LIN {X 0,Y 355.905,Z 472.152,A -85,B 0,C 180,E1 -13283.259,E2 -13283.259} C_VEL
LIN {X 0,Y 354.805,Z 472.289,A -85,B 0,C 180,E1 -13284.204,E2 -13284.204} C_VEL
LIN {X 0,Y 354.689,Z 472.301,A -85,B 0,C 180,E1 -13284.524,E2 -13284.524} C_VEL
LIN {X 0,Y 354.395,Z 472.343,A -85,B 0,C 180,E1 -13287.626,E2 -13287.626} C_VEL
LIN {X 0,Y 353.979,Z 472.396,A -85,B 0,C 180,E1 -13291.542,E2 -13291.542} C_VEL
LIN {X 0,Y 353.842,Z 472.551,A -85,B 0,C 180,E1 -13292.817,E2 -13292.817} C_VEL
LIN {X 0,Y 353.738,Z 476.121,A -85,B 0,C 180,E1 -13296.587,E2 -13296.587} C_VEL
LIN {X 0,Y 353.621,Z 479.721,A -85,B 0,C 180,E1 -13300.253,E2 -13300.253} C_VEL
LIN {X 0,Y 353.632,Z 480.392,A -85,B 0,C 180,E1 -13300.924,E2 -13300.924} C_VEL
LIN {X 0,Y 356.212,Z 492.931,A -85,B 0,C 180,E1 -13301.598,E2 -13301.598} C_VEL
LIN {X 0,Y 359.042,Z 506.674,A -85,B 0,C 180,E1 -13302.568,E2 -13302.568} C_VEL
LIN {X 0,Y 358.364,Z 517.999,A -85,B 0,C 180,E1 -13303.479,E2 -13303.479} C_VEL
LIN {X 0,Y 357.519,Z 529.506,A -85,B 0,C 180,E1 -13304.642,E2 -13304.642} C_VEL
LIN {X 0,Y 356.647,Z 540.627,A -85,B 0,C 180,E1 -13306.031,E2 -13306.031} C_VEL
LIN {X 0,Y 355.769,Z 549.851,A -85,B 0,C 180,E1 -13307.449,E2 -13307.449} C_VEL
LIN {X 0,Y 355.032,Z 558.925,A -85,B 0,C 180,E1 -13309.16,E2 -13309.16} C_VEL
LIN {X 0,Y 354.441,Z 566.279,A -85,B 0,C 180,E1 -13310.873,E2 -13310.873} C_VEL
LIN {X 0,Y 354.04,Z 572.161,A -85,B 0,C 180,E1 -13312.587,E2 -13312.587} C_VEL
LIN {X 0,Y 353.758,Z 576.815,A -85,B 0,C 180,E1 -13314.299,E2 -13314.299} C_VEL
LIN {X 0,Y 353.549,Z 580.37,A -85,B 0,C 180,E1 -13316.01,E2 -13316.01} C_VEL
LIN {X 0,Y 353.522,Z 582.903,A -85,B 0,C 180,E1 -13317.721,E2 -13317.721} C_VEL
LIN {X 0,Y 353.486,Z 584.043,A -85,B 0,C 180,E1 -13318.861,E2 -13318.861} C_VEL
LIN {X 0,Y 353.456,Z 584.785,A -85,B 0,C 180,E1 -13320,E2 -13320} C_VEL
LIN {X 0,Y 353.525,Z 585.12,A -85,B 0,C 180,E1 -13321.139,E2 -13321.139} C_VEL
LIN {X 0,Y 353.644,Z 585.007,A -85,B 0,C 180,E1 -13322.278,E2 -13322.278} C_VEL
LIN {X 0,Y 353.82,Z 584.499,A -85,B 0,C 180,E1 -13323.416,E2 -13323.416} C_VEL
LIN {X 0,Y 354.023,Z 583.603,A -85,B 0,C 180,E1 -13324.554,E2 -13324.554} C_VEL
LIN {X 0,Y 354.055,Z 582.303,A -85,B 0,C 180,E1 -13325.696,E2 -13325.696} C_VEL
LIN {X 0,Y 354.716,Z 578.614,A -85,B 0,C 180,E1 -13327.838,E2 -13327.838} C_VEL
LIN {X 0,Y 355.446,Z 574.19,A -85,B 0,C 180,E1 -13329.675,E2 -13329.675} C_VEL
LIN {X 0,Y 356.568,Z 567.89,A -85,B 0,C 180,E1 -13331.655,E2 -13331.655} C_VEL
LIN {X 0,Y 357.659,Z 561.049,A -85,B 0,C 180,E1 -13333.349,E2 -13333.349} C_VEL
LIN {X 0,Y 358.995,Z 552.647,A -85,B 0,C 180,E1 -13335.034,E2 -13335.034} C_VEL
LIN {X 0,Y 360.549,Z 544.142,A -85,B 0,C 180,E1 -13336.418,E2 -13336.418} C_VEL
LIN {X 0,Y 362.18,Z 532.806,A -85,B 0,C 180,E1 -13337.931,E2 -13337.931} C_VEL
LIN {X 0,Y 363.831,Z 521.052,A -85,B 0,C 180,E1 -13339.171,E2 -13339.171} C_VEL
LIN {X 0,Y 364.531,Z 514.204,A -85,B 0,C 180,E1 -13339.791,E2 -13339.791} C_VEL
LIN {X 0,Y 362.046,Z 504.538,A -85,B 0,C 180,E1 -13340.902,E2 -13340.902} C_VEL
LIN {X 0,Y 358.084,Z 494.328,A -85,B 0,C 180,E1 -13342.101,E2 -13342.101} C_VEL
LIN {X 0,Y 355.734,Z 489.62,A -85,B 0,C 180,E1 -13342.687,E2 -13342.687} C_VEL
LIN {X 0,Y 354.862,Z 487.017,A -85,B 0,C 180,E1 -13342.988,E2 -13342.988} C_VEL
LIN {X 0,Y 355.255,Z 485.091,A -85,B 0,C 180,E1 -13347.065,E2 -13347.065} C_VEL
LIN {X 0,Y 355.732,Z 483.771,A -85,B 0,C 180,E1 -13350.908,E2 -13350.908} C_VEL
LIN {X 0,Y 356.135,Z 483.121,A -85,B 0,C 180,E1 -13354.021,E2 -13354.021} C_VEL
LIN {X 0,Y 356.41,Z 482.934,A -85,B 0,C 180,E1 -13356.268,E2 -13356.268} C_VEL
LIN {X 0,Y 356.662,Z 483.11,A -85,B 0,C 180,E1 -13359.091,E2 -13359.091} C_VEL
LIN {X 0,Y 356.824,Z 483.837,A -85,B 0,C 180,E1 -13362.041,E2 -13362.041} C_VEL
LIN {X 0,Y 357.107,Z 485.188,A -85,B 0,C 180,E1 -13365.112,E2 -13365.112} C_VEL
LIN {X 0,Y 357.505,Z 487.296,A -85,B 0,C 180,E1 -13368.333,E2 -13368.333} C_VEL
LIN {X 0,Y 357.859,Z 490.386,A -85,B 0,C 180,E1 -13371.773,E2 -13371.773} C_VEL
LIN {X 0,Y 357.766,Z 492.788,A -85,B 0,C 180,E1 -13373.891,E2 -13373.891} C_VEL
LIN {X 0,Y 357.119,Z 496.371,A -85,B 0,C 180,E1 -13376.562,E2 -13376.562} C_VEL
LIN {X 0,Y 356.022,Z 502.317,A -85,B 0,C 180,E1 -13380.428,E2 -13380.428} C_VEL
LIN {X 0,Y 355.137,Z 508.799,A -85,B 0,C 180,E1 -13384.191,E2 -13384.191} C_VEL
LIN {X 0,Y 354.64,Z 514.033,A -85,B 0,C 180,E1 -13386.959,E2 -13386.959} C_VEL
LIN {X 0,Y 355.608,Z 517.659,A -85,B 0,C 180,E1 -13387.26,E2 -13387.26} C_VEL
LIN {X 0,Y 358.687,Z 529.151,A -85,B 0,C 180,E1 -13388.286,E2 -13388.286} C_VEL
LIN {X 0,Y 360.594,Z 540.569,A -85,B 0,C 180,E1 -13389.313,E2 -13389.313} C_VEL
LIN {X 0,Y 361.291,Z 549.72,A -85,B 0,C 180,E1 -13390.174,E2 -13390.174} C_VEL
LIN {X 0,Y 360.953,Z 561.989,A -85,B 0,C 180,E1 -13391.408,E2 -13391.408} C_VEL
LIN {X 0,Y 359.23,Z 574.08,A -85,B 0,C 180,E1 -13392.788,E2 -13392.788} C_VEL
LIN {X 0,Y 357.65,Z 584.49,A -85,B 0,C 180,E1 -13394.251,E2 -13394.251} C_VEL
LIN {X 0,Y 356.354,Z 593.147,A -85,B 0,C 180,E1 -13395.728,E2 -13395.728} C_VEL
LIN {X 0,Y 355.292,Z 601.393,A -85,B 0,C 180,E1 -13397.432,E2 -13397.432} C_VEL
LIN {X 0,Y 354.388,Z 608.162,A -85,B 0,C 180,E1 -13399.141,E2 -13399.141} C_VEL
LIN {X 0,Y 353.849,Z 613.658,A -85,B 0,C 180,E1 -13400.857,E2 -13400.857} C_VEL
LIN {X 0,Y 353.509,Z 618,A -85,B 0,C 180,E1 -13402.575,E2 -13402.575} C_VEL
LIN {X 0,Y 353.335,Z 621.292,A -85,B 0,C 180,E1 -13404.292,E2 -13404.292} C_VEL
LIN {X 0,Y 353.326,Z 622.934,A -85,B 0,C 180,E1 -13405.436,E2 -13405.436} C_VEL
LIN {X 0,Y 353.371,Z 624.929,A -85,B 0,C 180,E1 -13407.72,E2 -13407.72} C_VEL
LIN {X 0,Y 353.465,Z 625.318,A -85,B 0,C 180,E1 -13408.861,E2 -13408.861} C_VEL
LIN {X 0,Y 353.463,Z 625.241,A -85,B 0,C 180,E1 -13410,E2 -13410} C_VEL
LIN {X 0,Y 353.476,Z 624.735,A -85,B 0,C 180,E1 -13411.139,E2 -13411.139} C_VEL
LIN {X 0,Y 353.477,Z 623.816,A -85,B 0,C 180,E1 -13412.279,E2 -13412.279} C_VEL
LIN {X 0,Y 353.344,Z 622.452,A -85,B 0,C 180,E1 -13413.421,E2 -13413.421} C_VEL
LIN {X 0,Y 353.457,Z 619.538,A -85,B 0,C 180,E1 -13415.133,E2 -13415.133} C_VEL
LIN {X 0,Y 353.501,Z 615.509,A -85,B 0,C 180,E1 -13416.851,E2 -13416.851} C_VEL
LIN {X 0,Y 353.764,Z 609.258,A -85,B 0,C 180,E1 -13418.857,E2 -13418.857} C_VEL
LIN {X 0,Y 354.144,Z 602.428,A -85,B 0,C 180,E1 -13420.577,E2 -13420.577} C_VEL
LIN {X 0,Y 354.86,Z 593.944,A -85,B 0,C 180,E1 -13422.292,E2 -13422.292} C_VEL
LIN {X 0,Y 355.702,Z 583.664,A -85,B 0,C 180,E1 -13423.958,E2 -13423.958} C_VEL
LIN {X 0,Y 356.569,Z 573.529,A -85,B 0,C 180,E1 -13425.285,E2 -13425.285} C_VEL
LIN {X 0,Y 357.601,Z 561.386,A -85,B 0,C 180,E1 -13426.557,E2 -13426.557} C_VEL
LIN {X 0,Y 357.936,Z 554.907,A -85,B 0,C 180,E1 -13427.129,E2 -13427.129} C_VEL
LIN {X 0,Y 356.748,Z 542.906,A -85,B 0,C 180,E1 -13428.045,E2 -13428.045} C_VEL
LIN {X 0,Y 355.075,Z 528.958,A -85,B 0,C 180,E1 -13428.876,E2 -13428.876} C_VEL
LIN {X 0,Y 353.997,Z 519.742,A -85,B 0,C 180,E1 -13429.31,E2 -13429.31} C_VEL
LIN {X 0,Y 354.501,Z 511.518,A -85,B 0,C 180,E1 -13433.36,E2 -13433.36} C_VEL
LIN {X 0,Y 355.211,Z 504.084,A -85,B 0,C 180,E1 -13437.083,E2 -13437.083} C_VEL
LIN {X 0,Y 355.831,Z 497.874,A -85,B 0,C 180,E1 -13440.241,E2 -13440.241} C_VEL
LIN {X 0,Y 356.571,Z 491.594,A -85,B 0,C 180,E1 -13443.496,E2 -13443.496} C_VEL
LIN {X 0,Y 356.992,Z 487.823,A -85,B 0,C 180,E1 -13445.504,E2 -13445.504} C_VEL
LIN {X 0,Y 356.888,Z 483.993,A -85,B 0,C 180,E1 -13447.623,E2 -13447.623} C_VEL
LIN {X 0,Y 356.029,Z 478.756,A -85,B 0,C 180,E1 -13450.649,E2 -13450.649} C_VEL
LIN {X 0,Y 354.875,Z 472.282,A -85,B 0,C 180,E1 -13454.685,E2 -13454.685} C_VEL
LIN {X 0,Y 354.838,Z 472.282,A -85,B 0,C 180,E1 -13457.669,E2 -13457.669} C_VEL
LIN {X 0,Y 354.821,Z 472.289,A -85,B 0,C 180,E1 -13460.667,E2 -13460.667} C_VEL
LIN {X 0,Y 354.822,Z 472.287,A -85,B 0,C 180,E1 -13464.301,E2 -13464.301} C_VEL
LIN {X 0,Y 354.788,Z 472.288,A -85,B 0,C 180,E1 -13467.667,E2 -13467.667} C_VEL
LIN {X 0,Y 354.847,Z 472.281,A -85,B 0,C 180,E1 -13471.619,E2 -13471.619} C_VEL
LIN {X 0,Y 354.9,Z 472.276,A -85,B 0,C 180,E1 -13474.173,E2 -13474.173} C_VEL
LIN {X 0,Y 354.836,Z 472.283,A -85,B 0,C 180,E1 -13477.894,E2 -13477.894} C_VEL
LIN {X 0,Y 354.923,Z 472.272,A -85,B 0,C 180,E1 -13481.892,E2 -13481.892} C_VEL
LIN {X 0,Y 354.944,Z 472.27,A -85,B 0,C 180,E1 -13485.981,E2 -13485.981} C_VEL
LIN {X 0,Y 354.98,Z 472.264,A -85,B 0,C 180,E1 -13489.736,E2 -13489.736} C_VEL
LIN {X 0,Y 355.116,Z 472.249,A -85,B 0,C 180,E1 -13492.037,E2 -13492.037} C_VEL
LIN {X 0,Y 355.094,Z 472.255,A -85,B 0,C 180,E1 -13494.321,E2 -13494.321} C_VEL
LIN {X 0,Y 355.245,Z 472.231,A -85,B 0,C 180,E1 -13497.733,E2 -13497.733} C_VEL
LIN {X 0,Y 355.4,Z 472.214,A -85,B 0,C 180,E1 -13500,E2 -13500} C_VEL
LIN {X 0,Y 355.247,Z 472.235,A -85,B 0,C 180,E1 -13502.268,E2 -13502.268} C_VEL
LIN {X 0,Y 355.14,Z 472.248,A -85,B 0,C 180,E1 -13506.819,E2 -13506.819} C_VEL
LIN {X 0,Y 355.017,Z 472.261,A -85,B 0,C 180,E1 -13509.113,E2 -13509.113} C_VEL
LIN {X 0,Y 354.924,Z 472.276,A -85,B 0,C 180,E1 -13512.581,E2 -13512.581} C_VEL
LIN {X 0,Y 354.892,Z 472.279,A -85,B 0,C 180,E1 -13516.096,E2 -13516.096} C_VEL
LIN {X 0,Y 354.908,Z 472.278,A -85,B 0,C 180,E1 -13518.472,E2 -13518.472} C_VEL
LIN {X 0,Y 354.837,Z 472.286,A -85,B 0,C 180,E1 -13522.106,E2 -13522.106} C_VEL
LIN {X 0,Y 354.902,Z 472.276,A -85,B 0,C 180,E1 -13525.828,E2 -13525.828} C_VEL
LIN {X 0,Y 354.856,Z 472.281,A -85,B 0,C 180,E1 -13529.679,E2 -13529.679} C_VEL
LIN {X 0,Y 354.808,Z 472.286,A -85,B 0,C 180,E1 -13533.702,E2 -13533.702} C_VEL
LIN {X 0,Y 354.801,Z 472.292,A -85,B 0,C 180,E1 -13536.46,E2 -13536.46} C_VEL
LIN {X 0,Y 354.826,Z 472.284,A -85,B 0,C 180,E1 -13539.424,E2 -13539.424} C_VEL
LIN {X 0,Y 354.791,Z 472.289,A -85,B 0,C 180,E1 -13542.868,E2 -13542.868} C_VEL
LIN {X 0,Y 354.771,Z 472.295,A -85,B 0,C 180,E1 -13546.104,E2 -13546.104} C_VEL
LIN {X 0,Y 354.791,Z 472.288,A -85,B 0,C 180,E1 -13549.179,E2 -13549.179} C_VEL
LIN {X 0,Y 354.815,Z 472.289,A -85,B 0,C 180,E1 -13552.402,E2 -13552.402} C_VEL
LIN {X 0,Y 354.815,Z 472.285,A -85,B 0,C 180,E1 -13554.941,E2 -13554.941} C_VEL
LIN {X 0,Y 354.797,Z 472.292,A -85,B 0,C 180,E1 -13558.405,E2 -13558.405} C_VEL
LIN {X 0,Y 354.85,Z 472.282,A -85,B 0,C 180,E1 -13561.619,E2 -13561.619} C_VEL
LIN {X 0,Y 354.903,Z 472.279,A -85,B 0,C 180,E1 -13564.173,E2 -13564.173} C_VEL
LIN {X 0,Y 354.838,Z 472.286,A -85,B 0,C 180,E1 -13567.894,E2 -13567.894} C_VEL
LIN {X 0,Y 354.927,Z 472.275,A -85,B 0,C 180,E1 -13571.892,E2 -13571.892} C_VEL
LIN {X 0,Y 354.947,Z 472.273,A -85,B 0,C 180,E1 -13575.981,E2 -13575.981} C_VEL
LIN {X 0,Y 354.982,Z 472.267,A -85,B 0,C 180,E1 -13579.736,E2 -13579.736} C_VEL
LIN {X 0,Y 355.107,Z 472.249,A -85,B 0,C 180,E1 -13583.18,E2 -13583.18} C_VEL
LIN {X 0,Y 355.248,Z 472.235,A -85,B 0,C 180,E1 -13587.733,E2 -13587.733} C_VEL
LIN {X 0,Y 355.401,Z 472.217,A -85,B 0,C 180,E1 -13590,E2 -13590} C_VEL
LIN {X 0,Y 355.248,Z 472.235,A -85,B 0,C 180,E1 -13592.268,E2 -13592.268} C_VEL
LIN {X 0,Y 355.126,Z 472.246,A -85,B 0,C 180,E1 -13596.82,E2 -13596.82} C_VEL
LIN {X 0,Y 354.982,Z 472.267,A -85,B 0,C 180,E1 -13600.264,E2 -13600.264} C_VEL
LIN {X 0,Y 354.947,Z 472.274,A -85,B 0,C 180,E1 -13604.019,E2 -13604.019} C_VEL
LIN {X 0,Y 354.927,Z 472.275,A -85,B 0,C 180,E1 -13608.109,E2 -13608.109} C_VEL
LIN {X 0,Y 354.839,Z 472.286,A -85,B 0,C 180,E1 -13612.106,E2 -13612.106} C_VEL
LIN {X 0,Y 354.903,Z 472.279,A -85,B 0,C 180,E1 -13615.827,E2 -13615.827} C_VEL
LIN {X 0,Y 354.821,Z 472.288,A -85,B 0,C 180,E1 -13619.682,E2 -13619.682} C_VEL
LIN {X 0,Y 354.81,Z 472.291,A -85,B 0,C 180,E1 -13623.702,E2 -13623.702} C_VEL
LIN {X 0,Y 354.802,Z 472.287,A -85,B 0,C 180,E1 -13626.459,E2 -13626.459} C_VEL
LIN {X 0,Y 354.828,Z 472.286,A -85,B 0,C 180,E1 -13629.424,E2 -13629.424} C_VEL
LIN {X 0,Y 354.792,Z 472.288,A -85,B 0,C 180,E1 -13632.867,E2 -13632.867} C_VEL
LIN {X 0,Y 354.771,Z 472.293,A -85,B 0,C 180,E1 -13636.104,E2 -13636.104} C_VEL
LIN {X 0,Y 354.78,Z 472.288,A -85,B 0,C 180,E1 -13639.597,E2 -13639.597} C_VEL
LIN {X 0,Y 354.793,Z 472.288,A -85,B 0,C 180,E1 -13642.406,E2 -13642.406} C_VEL
LIN {X 0,Y 354.689,Z 472.301,A -85,B 0,C 180,E1 -13644.524,E2 -13644.524} C_VEL
LIN {X 0,Y 353.912,Z 472.402,A -85,B 0,C 180,E1 -13645.47,E2 -13645.47} C_VEL
LIN {X 0,Y 350.871,Z 472.777,A -85,B 0,C 180,E1 -13647.002,E2 -13647.002} C_VEL
LIN {X 0,Y 348.33,Z 473.095,A -85,B 0,C 180,E1 -13648.243,E2 -13648.243} C_VEL
LIN {X 0,Y 347.232,Z 473.232,A -85,B 0,C 180,E1 -13649.206,E2 -13649.206} C_VEL
LIN {X 0,Y 347.137,Z 473.246,A -85,B 0,C 180,E1 -13649.533,E2 -13649.533} C_VEL
LIN {X 0,Y 346.856,Z 473.284,A -85,B 0,C 180,E1 -13652.223,E2 -13652.223} C_VEL
LIN {X 0,Y 346.776,Z 473.898,A -85,B 0,C 180,E1 -13653.521,E2 -13653.521} C_VEL
LIN {X 0,Y 346.629,Z 477.509,A -85,B 0,C 180,E1 -13657.342,E2 -13657.342} C_VEL
LIN {X 0,Y 346.574,Z 480.732,A -85,B 0,C 180,E1 -13660.644,E2 -13660.644} C_VEL
LIN {X 0,Y 349.725,Z 496.151,A -85,B 0,C 180,E1 -13661.547,E2 -13661.547} C_VEL
LIN {X 0,Y 351.969,Z 507.166,A -85,B 0,C 180,E1 -13662.365,E2 -13662.365} C_VEL
LIN {X 0,Y 351.387,Z 518.382,A -85,B 0,C 180,E1 -13663.291,E2 -13663.291} C_VEL
LIN {X 0,Y 350.478,Z 530.384,A -85,B 0,C 180,E1 -13664.534,E2 -13664.534} C_VEL
LIN {X 0,Y 349.631,Z 541.006,A -85,B 0,C 180,E1 -13665.893,E2 -13665.893} C_VEL
LIN {X 0,Y 348.67,Z 551.064,A -85,B 0,C 180,E1 -13667.485,E2 -13667.485} C_VEL
LIN {X 0,Y 347.921,Z 560.021,A -85,B 0,C 180,E1 -13669.231,E2 -13669.231} C_VEL
LIN {X 0,Y 347.303,Z 567.219,A -85,B 0,C 180,E1 -13670.977,E2 -13670.977} C_VEL
LIN {X 0,Y 346.895,Z 574.058,A -85,B 0,C 180,E1 -13673.088,E2 -13673.088} C_VEL
LIN {X 0,Y 346.625,Z 578.231,A -85,B 0,C 180,E1 -13674.765,E2 -13674.765} C_VEL
LIN {X 0,Y 346.443,Z 581.525,A -85,B 0,C 180,E1 -13676.511,E2 -13676.511} C_VEL
LIN {X 0,Y 346.428,Z 583.179,A -85,B 0,C 180,E1 -13677.674,E2 -13677.674} C_VEL
LIN {X 0,Y 346.406,Z 584.367,A -85,B 0,C 180,E1 -13678.837,E2 -13678.837} C_VEL
LIN {X 0,Y 346.463,Z 585.56,A -85,B 0,C 180,E1 -13681.162,E2 -13681.162} C_VEL
LIN {X 0,Y 346.589,Z 585.527,A -85,B 0,C 180,E1 -13682.324,E2 -13682.324} C_VEL
LIN {X 0,Y 346.777,Z 585.066,A -85,B 0,C 180,E1 -13683.486,E2 -13683.486} C_VEL
LIN {X 0,Y 346.985,Z 584.216,A -85,B 0,C 180,E1 -13684.647,E2 -13684.647} C_VEL
LIN {X 0,Y 347.018,Z 583,A -85,B 0,C 180,E1 -13685.812,E2 -13685.812} C_VEL
LIN {X 0,Y 347.734,Z 579.51,A -85,B 0,C 180,E1 -13687.971,E2 -13687.971} C_VEL
LIN {X 0,Y 348.515,Z 575.157,A -85,B 0,C 180,E1 -13689.87,E2 -13689.87} C_VEL
LIN {X 0,Y 349.535,Z 569.974,A -85,B 0,C 180,E1 -13691.599,E2 -13691.599} C_VEL
LIN {X 0,Y 350.66,Z 563.577,A -85,B 0,C 180,E1 -13693.326,E2 -13693.326} C_VEL
LIN {X 0,Y 352.016,Z 555.705,A -85,B 0,C 180,E1 -13695.043,E2 -13695.043} C_VEL
LIN {X 0,Y 353.919,Z 545.903,A -85,B 0,C 180,E1 -13696.734,E2 -13696.734} C_VEL
LIN {X 0,Y 355.665,Z 534.941,A -85,B 0,C 180,E1 -13698.271,E2 -13698.271} C_VEL
LIN {X 0,Y 357.401,Z 523.779,A -85,B 0,C 180,E1 -13699.529,E2 -13699.529} C_VEL
LIN {X 0,Y 358.27,Z 516.092,A -85,B 0,C 180,E1 -13700.267,E2 -13700.267} C_VEL
LIN {X 0,Y 355.81,Z 506.506,A -85,B 0,C 180,E1 -13701.438,E2 -13701.438} C_VEL
LIN {X 0,Y 351.844,Z 496.555,A -85,B 0,C 180,E1 -13702.714,E2 -13702.714} C_VEL
LIN {X 0,Y 348.086,Z 488.614,A -85,B 0,C 180,E1 -13703.767,E2 -13703.767} C_VEL
LIN {X 0,Y 347.924,Z 487.83,A -85,B 0,C 180,E1 -13703.881,E2 -13703.881} C_VEL
LIN {X 0,Y 348.332,Z 486.201,A -85,B 0,C 180,E1 -13707.649,E2 -13707.649} C_VEL
LIN {X 0,Y 348.674,Z 485.347,A -85,B 0,C 180,E1 -13710.259,E2 -13710.259} C_VEL
LIN {X 0,Y 349.039,Z 484.766,A -85,B 0,C 180,E1 -13712.933,E2 -13712.933} C_VEL
LIN {X 0,Y 349.504,Z 484.446,A -85,B 0,C 180,E1 -13716.453,E2 -13716.453} C_VEL
LIN {X 0,Y 349.681,Z 484.569,A -85,B 0,C 180,E1 -13718.539,E2 -13718.539} C_VEL
LIN {X 0,Y 349.878,Z 485.222,A -85,B 0,C 180,E1 -13721.519,E2 -13721.519} C_VEL
LIN {X 0,Y 350.123,Z 486.493,A -85,B 0,C 180,E1 -13724.632,E2 -13724.632} C_VEL
LIN {X 0,Y 350.518,Z 488.505,A -85,B 0,C 180,E1 -13727.89,E2 -13727.89} C_VEL
LIN {X 0,Y 350.878,Z 491.474,A -85,B 0,C 180,E1 -13731.367,E2 -13731.367} C_VEL
LIN {X 0,Y 350.864,Z 493.475,A -85,B 0,C 180,E1 -13733.247,E2 -13733.247} C_VEL
LIN {X 0,Y 350.355,Z 496.731,A -85,B 0,C 180,E1 -13735.828,E2 -13735.828} C_VEL
LIN {X 0,Y 349.373,Z 501.511,A -85,B 0,C 180,E1 -13739.139,E2 -13739.139} C_VEL
LIN {X 0,Y 348.496,Z 506.982,A -85,B 0,C 180,E1 -13742.54,E2 -13742.54} C_VEL
LIN {X 0,Y 347.767,Z 513.422,A -85,B 0,C 180,E1 -13746.086,E2 -13746.086} C_VEL
LIN {X 0,Y 348.764,Z 516.99,A -85,B 0,C 180,E1 -13746.418,E2 -13746.418} C_VEL
LIN {X 0,Y 352.237,Z 529.577,A -85,B 0,C 180,E1 -13747.637,E2 -13747.637} C_VEL
LIN {X 0,Y 354.251,Z 541.8,A -85,B 0,C 180,E1 -13748.818,E2 -13748.818} C_VEL
LIN {X 0,Y 354.883,Z 550.961,A -85,B 0,C 180,E1 -13749.728,E2 -13749.728} C_VEL
LIN {X 0,Y 354.52,Z 562.022,A -85,B 0,C 180,E1 -13750.907,E2 -13750.907} C_VEL
LIN {X 0,Y 352.685,Z 573.949,A -85,B 0,C 180,E1 -13752.308,E2 -13752.308} C_VEL
LIN {X 0,Y 351.074,Z 583.779,A -85,B 0,C 180,E1 -13753.724,E2 -13753.724} C_VEL
LIN {X 0,Y 349.694,Z 592.06,A -85,B 0,C 180,E1 -13755.153,E2 -13755.153} C_VEL
LIN {X 0,Y 348.55,Z 600.362,A -85,B 0,C 180,E1 -13756.889,E2 -13756.889} C_VEL
LIN {X 0,Y 347.371,Z 608.231,A -85,B 0,C 180,E1 -13758.918,E2 -13758.918} C_VEL
LIN {X 0,Y 346.819,Z 613.593,A -85,B 0,C 180,E1 -13760.67,E2 -13760.67} C_VEL
LIN {X 0,Y 346.442,Z 617.838,A -85,B 0,C 180,E1 -13762.423,E2 -13762.423} C_VEL
LIN {X 0,Y 346.249,Z 621.052,A -85,B 0,C 180,E1 -13764.175,E2 -13764.175} C_VEL
LIN {X 0,Y 346.239,Z 622.623,A -85,B 0,C 180,E1 -13765.343,E2 -13765.343} C_VEL
LIN {X 0,Y 346.216,Z 623.784,A -85,B 0,C 180,E1 -13766.508,E2 -13766.508} C_VEL
LIN {X 0,Y 346.272,Z 624.542,A -85,B 0,C 180,E1 -13767.673,E2 -13767.673} C_VEL
LIN {X 0,Y 346.4,Z 624.87,A -85,B 0,C 180,E1 -13768.837,E2 -13768.837} C_VEL
LIN {X 0,Y 346.399,Z 624.738,A -85,B 0,C 180,E1 -13770,E2 -13770} C_VEL
LIN {X 0,Y 346.414,Z 624.196,A -85,B 0,C 180,E1 -13771.162,E2 -13771.162} C_VEL
LIN {X 0,Y 346.397,Z 623.234,A -85,B 0,C 180,E1 -13772.325,E2 -13772.325} C_VEL
LIN {X 0,Y 346.266,Z 621.79,A -85,B 0,C 180,E1 -13773.491,E2 -13773.491} C_VEL
LIN {X 0,Y 346.373,Z 618.794,A -85,B 0,C 180,E1 -13775.239,E2 -13775.239} C_VEL
LIN {X 0,Y 346.417,Z 614.67,A -85,B 0,C 180,E1 -13776.992,E2 -13776.992} C_VEL
LIN {X 0,Y 346.703,Z 608.322,A -85,B 0,C 180,E1 -13779.038,E2 -13779.038} C_VEL
LIN {X 0,Y 347.115,Z 601.385,A -85,B 0,C 180,E1 -13780.794,E2 -13780.794} C_VEL
LIN {X 0,Y 347.883,Z 592.728,A -85,B 0,C 180,E1 -13782.543,E2 -13782.543} C_VEL
LIN {X 0,Y 348.704,Z 582.564,A -85,B 0,C 180,E1 -13784.201,E2 -13784.201} C_VEL
LIN {X 0,Y 349.674,Z 571.893,A -85,B 0,C 180,E1 -13785.594,E2 -13785.594} C_VEL
LIN {X 0,Y 350.704,Z 559.503,A -85,B 0,C 180,E1 -13786.892,E2 -13786.892} C_VEL
LIN {X 0,Y 350.831,Z 554.51,A -85,B 0,C 180,E1 -13787.336,E2 -13787.336} C_VEL
LIN {X 0,Y 349.545,Z 542.138,A -85,B 0,C 180,E1 -13788.303,E2 -13788.303} C_VEL
LIN {X 0,Y 347.932,Z 528.31,A -85,B 0,C 180,E1 -13789.143,E2 -13789.143} C_VEL
LIN {X 0,Y 346.911,Z 519.419,A -85,B 0,C 180,E1 -13789.567,E2 -13789.567} C_VEL
LIN {X 0,Y 347.4,Z 512.16,A -85,B 0,C 180,E1 -13793.234,E2 -13793.234} C_VEL
LIN {X 0,Y 347.963,Z 506.001,A -85,B 0,C 180,E1 -13796.381,E2 -13796.381} C_VEL
LIN {X 0,Y 348.716,Z 499.158,A -85,B 0,C 180,E1 -13799.932,E2 -13799.932} C_VEL
LIN {X 0,Y 349.533,Z 492.319,A -85,B 0,C 180,E1 -13803.569,E2 -13803.569} C_VEL
LIN {X 0,Y 349.969,Z 488.545,A -85,B 0,C 180,E1 -13805.618,E2 -13805.618} C_VEL
LIN {X 0,Y 349.84,Z 484.83,A -85,B 0,C 180,E1 -13807.705,E2 -13807.705} C_VEL
LIN {X 0,Y 348.942,Z 479.479,A -85,B 0,C 180,E1 -13810.887,E2 -13810.887} C_VEL
LIN {X 0,Y 347.842,Z 473.158,A -85,B 0,C 180,E1 -13814.9,E2 -13814.9} C_VEL
LIN {X 0,Y 347.785,Z 473.164,A -85,B 0,C 180,E1 -13818.391,E2 -13818.391} C_VEL
LIN {X 0,Y 347.774,Z 473.162,A -85,B 0,C 180,E1 -13822.011,E2 -13822.011} C_VEL
LIN {X 0,Y 347.745,Z 473.166,A -85,B 0,C 180,E1 -13825.536,E2 -13825.536} C_VEL
LIN {X 0,Y 347.746,Z 473.168,A -85,B 0,C 180,E1 -13828.301,E2 -13828.301} C_VEL
LIN {X 0,Y 347.779,Z 473.164,A -85,B 0,C 180,E1 -13830.988,E2 -13830.988} C_VEL
LIN {X 0,Y 347.832,Z 473.155,A -85,B 0,C 180,E1 -13833.608,E2 -13833.608} C_VEL
LIN {X 0,Y 347.79,Z 473.161,A -85,B 0,C 180,E1 -13836.162,E2 -13836.162} C_VEL
LIN {X 0,Y 347.814,Z 473.158,A -85,B 0,C 180,E1 -13839.909,E2 -13839.909} C_VEL
LIN {X 0,Y 347.867,Z 473.154,A -85,B 0,C 180,E1 -13842.359,E2 -13842.359} C_VEL
LIN {X 0,Y 347.898,Z 473.148,A -85,B 0,C 180,E1 -13845.971,E2 -13845.971} C_VEL
LIN {X 0,Y 347.93,Z 473.142,A -85,B 0,C 180,E1 -13849.526,E2 -13849.526} C_VEL
LIN {X 0,Y 348.076,Z 473.125,A -85,B 0,C 180,E1 -13851.875,E2 -13851.875} C_VEL
LIN {X 0,Y 348.069,Z 473.128,A -85,B 0,C 180,E1 -13854.206,E2 -13854.206} C_VEL
LIN {X 0,Y 348.208,Z 473.108,A -85,B 0,C 180,E1 -13857.687,E2 -13857.687} C_VEL
LIN {X 0,Y 348.348,Z 473.092,A -85,B 0,C 180,E1 -13860,E2 -13860} C_VEL
LIN {X 0,Y 348.21,Z 473.112,A -85,B 0,C 180,E1 -13862.314,E2 -13862.314} C_VEL
LIN {X 0,Y 348.108,Z 473.122,A -85,B 0,C 180,E1 -13866.958,E2 -13866.958} C_VEL
LIN {X 0,Y 347.969,Z 473.138,A -85,B 0,C 180,E1 -13869.299,E2 -13869.299} C_VEL
LIN {X 0,Y 347.892,Z 473.15,A -85,B 0,C 180,E1 -13872.84,E2 -13872.84} C_VEL
LIN {X 0,Y 347.841,Z 473.159,A -85,B 0,C 180,E1 -13876.432,E2 -13876.432} C_VEL
LIN {X 0,Y 347.858,Z 473.153,A -85,B 0,C 180,E1 -13878.86,E2 -13878.86} C_VEL
LIN {X 0,Y 347.776,Z 473.166,A -85,B 0,C 180,E1 -13882.58,E2 -13882.58} C_VEL
LIN {X 0,Y 347.814,Z 473.157,A -85,B 0,C 180,E1 -13885.109,E2 -13885.109} C_VEL
LIN {X 0,Y 347.813,Z 473.158,A -85,B 0,C 180,E1 -13887.694,E2 -13887.694} C_VEL
LIN {X 0,Y 347.766,Z 473.168,A -85,B 0,C 180,E1 -13890.347,E2 -13890.347} C_VEL
LIN {X 0,Y 347.747,Z 473.17,A -85,B 0,C 180,E1 -13894.464,E2 -13894.464} C_VEL
LIN {X 0,Y 347.776,Z 473.165,A -85,B 0,C 180,E1 -13897.989,E2 -13897.989} C_VEL
LIN {X 0,Y 347.753,Z 473.166,A -85,B 0,C 180,E1 -13901.83,E2 -13901.83} C_VEL
LIN {X 0,Y 347.71,Z 473.17,A -85,B 0,C 180,E1 -13905.027,E2 -13905.027} C_VEL
LIN {X 0,Y 347.753,Z 473.169,A -85,B 0,C 180,E1 -13908.397,E2 -13908.397} C_VEL
LIN {X 0,Y 347.78,Z 473.166,A -85,B 0,C 180,E1 -13912.011,E2 -13912.011} C_VEL
LIN {X 0,Y 347.747,Z 473.166,A -85,B 0,C 180,E1 -13915.536,E2 -13915.536} C_VEL
LIN {X 0,Y 347.748,Z 473.17,A -85,B 0,C 180,E1 -13918.301,E2 -13918.301} C_VEL
LIN {X 0,Y 347.782,Z 473.161,A -85,B 0,C 180,E1 -13920.988,E2 -13920.988} C_VEL
LIN {X 0,Y 347.834,Z 473.156,A -85,B 0,C 180,E1 -13923.608,E2 -13923.608} C_VEL
LIN {X 0,Y 347.792,Z 473.165,A -85,B 0,C 180,E1 -13926.162,E2 -13926.162} C_VEL
LIN {X 0,Y 347.821,Z 473.16,A -85,B 0,C 180,E1 -13929.91,E2 -13929.91} C_VEL
LIN {X 0,Y 347.87,Z 473.154,A -85,B 0,C 180,E1 -13932.36,E2 -13932.36} C_VEL
LIN {X 0,Y 347.901,Z 473.151,A -85,B 0,C 180,E1 -13935.971,E2 -13935.971} C_VEL
LIN {X 0,Y 347.933,Z 473.144,A -85,B 0,C 180,E1 -13939.526,E2 -13939.526} C_VEL
LIN {X 0,Y 348.075,Z 473.124,A -85,B 0,C 180,E1 -13943.042,E2 -13943.042} C_VEL
LIN {X 0,Y 348.21,Z 473.111,A -85,B 0,C 180,E1 -13947.687,E2 -13947.687} C_VEL
LIN {X 0,Y 348.349,Z 473.096,A -85,B 0,C 180,E1 -13950,E2 -13950} C_VEL
LIN {X 0,Y 348.211,Z 473.111,A -85,B 0,C 180,E1 -13952.314,E2 -13952.314} C_VEL
LIN {X 0,Y 348.093,Z 473.122,A -85,B 0,C 180,E1 -13956.958,E2 -13956.958} C_VEL
LIN {X 0,Y 347.933,Z 473.144,A -85,B 0,C 180,E1 -13960.474,E2 -13960.474} C_VEL
LIN {X 0,Y 347.903,Z 473.15,A -85,B 0,C 180,E1 -13964.15,E2 -13964.15} C_VEL
LIN {X 0,Y 347.896,Z 473.149,A -85,B 0,C 180,E1 -13968.291,E2 -13968.291} C_VEL
LIN {X 0,Y 347.793,Z 473.163,A -85,B 0,C 180,E1 -13971.635,E2 -13971.635} C_VEL
LIN {X 0,Y 347.816,Z 473.157,A -85,B 0,C 180,E1 -13975.108,E2 -13975.108} C_VEL
LIN {X 0,Y 347.812,Z 473.162,A -85,B 0,C 180,E1 -13977.694,E2 -13977.694} C_VEL
LIN {X 0,Y 347.753,Z 473.166,A -85,B 0,C 180,E1 -13980.348,E2 -13980.348} C_VEL
LIN {X 0,Y 347.752,Z 473.169,A -85,B 0,C 180,E1 -13984.044,E2 -13984.044} C_VEL
LIN {X 0,Y 347.766,Z 473.165,A -85,B 0,C 180,E1 -13987.321,E2 -13987.321} C_VEL
LIN {X 0,Y 347.736,Z 473.168,A -85,B 0,C 180,E1 -13990.297,E2 -13990.297} C_VEL
LIN {X 0,Y 347.726,Z 473.171,A -85,B 0,C 180,E1 -13993.408,E2 -13993.408} C_VEL
LIN {X 0,Y 347.728,Z 473.168,A -85,B 0,C 180,E1 -13996.686,E2 -13996.686} C_VEL
LIN {X 0,Y 347.751,Z 473.167,A -85,B 0,C 180,E1 -14000.173,E2 -14000.173} C_VEL
LIN {X 0,Y 347.74,Z 473.166,A -85,B 0,C 180,E1 -14002.676,E2 -14002.676} C_VEL
LIN {X 0,Y 347.493,Z 473.2,A -85,B 0,C 180,E1 -14006.019,E2 -14006.019} C_VEL
LIN {X 0,Y 347.137,Z 473.246,A -85,B 0,C 180,E1 -14009.533,E2 -14009.533} C_VEL
LIN {X 0,Y 346.414,Z 473.337,A -85,B 0,C 180,E1 -14010.5,E2 -14010.5} C_VEL
LIN {X 0,Y 343.397,Z 473.824,A -85,B 0,C 180,E1 -14012.068,E2 -14012.068} C_VEL
LIN {X 0,Y 340.842,Z 474.55,A -85,B 0,C 180,E1 -14013.333,E2 -14013.333} C_VEL
LIN {X 0,Y 339.73,Z 475.313,A -85,B 0,C 180,E1 -14014.311,E2 -14014.311} C_VEL
LIN {X 0,Y 339.632,Z 475.612,A -85,B 0,C 180,E1 -14014.642,E2 -14014.642} C_VEL
LIN {X 0,Y 339.538,Z 479.417,A -85,B 0,C 180,E1 -14018.661,E2 -14018.661} C_VEL
LIN {X 0,Y 339.513,Z 481.32,A -85,B 0,C 180,E1 -14020.422,E2 -14020.422} C_VEL
LIN {X 0,Y 342.117,Z 493.902,A -85,B 0,C 180,E1 -14021.13,E2 -14021.13} C_VEL
LIN {X 0,Y 344.806,Z 507.157,A -85,B 0,C 180,E1 -14022.112,E2 -14022.112} C_VEL
LIN {X 0,Y 345.006,Z 510.206,A -85,B 0,C 180,E1 -14022.361,E2 -14022.361} C_VEL
LIN {X 0,Y 344.139,Z 521.771,A -85,B 0,C 180,E1 -14023.387,E2 -14023.387} C_VEL
LIN {X 0,Y 343.352,Z 532.499,A -85,B 0,C 180,E1 -14024.568,E2 -14024.568} C_VEL
LIN {X 0,Y 342.383,Z 543.313,A -85,B 0,C 180,E1 -14026.043,E2 -14026.043} C_VEL
LIN {X 0,Y 341.553,Z 552.222,A -85,B 0,C 180,E1 -14027.522,E2 -14027.522} C_VEL
LIN {X 0,Y 340.797,Z 561.012,A -85,B 0,C 180,E1 -14029.304,E2 -14029.304} C_VEL
LIN {X 0,Y 340.164,Z 568.083,A -85,B 0,C 180,E1 -14031.086,E2 -14031.086} C_VEL
LIN {X 0,Y 339.771,Z 574.583,A -85,B 0,C 180,E1 -14033.15,E2 -14033.15} C_VEL
LIN {X 0,Y 339.487,Z 579.545,A -85,B 0,C 180,E1 -14035.25,E2 -14035.25} C_VEL
LIN {X 0,Y 339.36,Z 581.692,A -85,B 0,C 180,E1 -14036.438,E2 -14036.438} C_VEL
LIN {X 0,Y 339.334,Z 583.419,A -85,B 0,C 180,E1 -14037.626,E2 -14037.626} C_VEL
LIN {X 0,Y 339.329,Z 584.692,A -85,B 0,C 180,E1 -14038.813,E2 -14038.813} C_VEL
LIN {X 0,Y 339.332,Z 585.536,A -85,B 0,C 180,E1 -14040,E2 -14040} C_VEL
LIN {X 0,Y 339.403,Z 585.986,A -85,B 0,C 180,E1 -14041.186,E2 -14041.186} C_VEL
LIN {X 0,Y 339.536,Z 586.038,A -85,B 0,C 180,E1 -14042.372,E2 -14042.372} C_VEL
LIN {X 0,Y 339.736,Z 585.647,A -85,B 0,C 180,E1 -14043.558,E2 -14043.558} C_VEL
LIN {X 0,Y 339.949,Z 584.859,A -85,B 0,C 180,E1 -14044.743,E2 -14044.743} C_VEL
LIN {X 0,Y 339.985,Z 583.705,A -85,B 0,C 180,E1 -14045.932,E2 -14045.932} C_VEL
LIN {X 0,Y 340.317,Z 582.119,A -85,B 0,C 180,E1 -14047.118,E2 -14047.118} C_VEL
LIN {X 0,Y 341.118,Z 578.874,A -85,B 0,C 180,E1 -14048.889,E2 -14048.889} C_VEL
LIN {X 0,Y 341.852,Z 574.631,A -85,B 0,C 180,E1 -14050.663,E2 -14050.663} C_VEL
LIN {X 0,Y 343.241,Z 568.183,A -85,B 0,C 180,E1 -14052.715,E2 -14052.715} C_VEL
LIN {X 0,Y 344.643,Z 561.248,A -85,B 0,C 180,E1 -14054.466,E2 -14054.466} C_VEL
LIN {X 0,Y 345.972,Z 554.264,A -85,B 0,C 180,E1 -14055.916,E2 -14055.916} C_VEL
LIN {X 0,Y 347.69,Z 545.994,A -85,B 0,C 180,E1 -14057.346,E2 -14057.346} C_VEL
LIN {X 0,Y 349.391,Z 536.056,A -85,B 0,C 180,E1 -14058.774,E2 -14058.774} C_VEL
LIN {X 0,Y 351.419,Z 523.79,A -85,B 0,C 180,E1 -14060.179,E2 -14060.179} C_VEL
LIN {X 0,Y 352.07,Z 518.155,A -85,B 0,C 180,E1 -14060.747,E2 -14060.747} C_VEL
LIN {X 0,Y 349.649,Z 508.549,A -85,B 0,C 180,E1 -14062.009,E2 -14062.009} C_VEL
LIN {X 0,Y 345.69,Z 498.633,A -85,B 0,C 180,E1 -14063.392,E2 -14063.392} C_VEL
LIN {X 0,Y 341.145,Z 489.171,A -85,B 0,C 180,E1 -14064.761,E2 -14064.761} C_VEL
LIN {X 0,Y 341.042,Z 488.678,A -85,B 0,C 180,E1 -14064.821,E2 -14064.821} C_VEL
LIN {X 0,Y 341.439,Z 487.355,A -85,B 0,C 180,E1 -14068.256,E2 -14068.256} C_VEL
LIN {X 0,Y 341.804,Z 486.599,A -85,B 0,C 180,E1 -14070.933,E2 -14070.933} C_VEL
LIN {X 0,Y 342.172,Z 486.113,A -85,B 0,C 180,E1 -14073.681,E2 -14073.681} C_VEL
LIN {X 0,Y 342.601,Z 485.971,A -85,B 0,C 180,E1 -14076.866,E2 -14076.866} C_VEL
LIN {X 0,Y 342.811,Z 486.283,A -85,B 0,C 180,E1 -14079.46,E2 -14079.46} C_VEL
LIN {X 0,Y 343.017,Z 487.156,A -85,B 0,C 180,E1 -14082.542,E2 -14082.542} C_VEL
LIN {X 0,Y 343.347,Z 488.754,A -85,B 0,C 180,E1 -14085.897,E2 -14085.897} C_VEL
LIN {X 0,Y 343.706,Z 491.042,A -85,B 0,C 180,E1 -14089.162,E2 -14089.162} C_VEL
LIN {X 0,Y 343.926,Z 493.817,A -85,B 0,C 180,E1 -14092.19,E2 -14092.19} C_VEL
LIN {X 0,Y 343.585,Z 496.936,A -85,B 0,C 180,E1 -14094.905,E2 -14094.905} C_VEL
LIN {X 0,Y 342.729,Z 500.807,A -85,B 0,C 180,E1 -14097.781,E2 -14097.781} C_VEL
LIN {X 0,Y 341.818,Z 505.798,A -85,B 0,C 180,E1 -14101.107,E2 -14101.107} C_VEL
LIN {X 0,Y 340.901,Z 512.51,A -85,B 0,C 180,E1 -14105.108,E2 -14105.108} C_VEL
LIN {X 0,Y 341.818,Z 516.036,A -85,B 0,C 180,E1 -14105.444,E2 -14105.444} C_VEL
LIN {X 0,Y 342.653,Z 518.554,A -85,B 0,C 180,E1 -14105.717,E2 -14105.717} C_VEL
LIN {X 0,Y 345.798,Z 529.963,A -85,B 0,C 180,E1 -14106.937,E2 -14106.937} C_VEL
LIN {X 0,Y 347.857,Z 542.251,A -85,B 0,C 180,E1 -14108.208,E2 -14108.208} C_VEL
LIN {X 0,Y 348.471,Z 552.117,A -85,B 0,C 180,E1 -14109.256,E2 -14109.256} C_VEL
LIN {X 0,Y 347.954,Z 563.564,A -85,B 0,C 180,E1 -14110.533,E2 -14110.533} C_VEL
LIN {X 0,Y 346.178,Z 573.951,A -85,B 0,C 180,E1 -14111.812,E2 -14111.812} C_VEL
LIN {X 0,Y 344.324,Z 584.481,A -85,B 0,C 180,E1 -14113.396,E2 -14113.396} C_VEL
LIN {X 0,Y 342.635,Z 594.026,A -85,B 0,C 180,E1 -14115.144,E2 -14115.144} C_VEL
LIN {X 0,Y 341.45,Z 601.864,A -85,B 0,C 180,E1 -14116.914,E2 -14116.914} C_VEL
LIN {X 0,Y 340.384,Z 608.308,A -85,B 0,C 180,E1 -14118.688,E2 -14118.688} C_VEL
LIN {X 0,Y 339.772,Z 613.544,A -85,B 0,C 180,E1 -14120.475,E2 -14120.475} C_VEL
LIN {X 0,Y 339.379,Z 617.681,A -85,B 0,C 180,E1 -14122.264,E2 -14122.264} C_VEL
LIN {X 0,Y 339.17,Z 620.798,A -85,B 0,C 180,E1 -14124.053,E2 -14124.053} C_VEL
LIN {X 0,Y 339.136,Z 622.323,A -85,B 0,C 180,E1 -14125.245,E2 -14125.245} C_VEL
LIN {X 0,Y 339.137,Z 623.443,A -85,B 0,C 180,E1 -14126.436,E2 -14126.436} C_VEL
LIN {X 0,Y 339.176,Z 624.148,A -85,B 0,C 180,E1 -14127.625,E2 -14127.625} C_VEL
LIN {X 0,Y 339.335,Z 624.401,A -85,B 0,C 180,E1 -14128.813,E2 -14128.813} C_VEL
LIN {X 0,Y 339.338,Z 624.229,A -85,B 0,C 180,E1 -14130,E2 -14130} C_VEL
LIN {X 0,Y 339.353,Z 623.644,A -85,B 0,C 180,E1 -14131.187,E2 -14131.187} C_VEL
LIN {X 0,Y 339.304,Z 622.619,A -85,B 0,C 180,E1 -14132.374,E2 -14132.374} C_VEL
LIN {X 0,Y 339.19,Z 621.107,A -85,B 0,C 180,E1 -14133.564,E2 -14133.564} C_VEL
LIN {X 0,Y 339.294,Z 618.022,A -85,B 0,C 180,E1 -14135.348,E2 -14135.348} C_VEL
LIN {X 0,Y 339.367,Z 613.806,A -85,B 0,C 180,E1 -14137.138,E2 -14137.138} C_VEL
LIN {X 0,Y 339.653,Z 607.35,A -85,B 0,C 180,E1 -14139.228,E2 -14139.228} C_VEL
LIN {X 0,Y 340.082,Z 600.238,A -85,B 0,C 180,E1 -14141.02,E2 -14141.02} C_VEL
LIN {X 0,Y 340.872,Z 591.426,A -85,B 0,C 180,E1 -14142.805,E2 -14142.805} C_VEL
LIN {X 0,Y 341.635,Z 582.445,A -85,B 0,C 180,E1 -14144.292,E2 -14144.292} C_VEL
LIN {X 0,Y 342.671,Z 571.41,A -85,B 0,C 180,E1 -14145.768,E2 -14145.768} C_VEL
LIN {X 0,Y 343.723,Z 559.042,A -85,B 0,C 180,E1 -14147.093,E2 -14147.093} C_VEL
LIN {X 0,Y 343.72,Z 554.009,A -85,B 0,C 180,E1 -14147.553,E2 -14147.553} C_VEL
LIN {X 0,Y 342.311,Z 540.955,A -85,B 0,C 180,E1 -14148.588,E2 -14148.588} C_VEL
LIN {X 0,Y 340.733,Z 527.25,A -85,B 0,C 180,E1 -14149.426,E2 -14149.426} C_VEL
LIN {X 0,Y 339.851,Z 519.076,A -85,B 0,C 180,E1 -14149.833,E2 -14149.833} C_VEL
LIN {X 0,Y 340.395,Z 511.541,A -85,B 0,C 180,E1 -14153.741,E2 -14153.741} C_VEL
LIN {X 0,Y 341.195,Z 504.092,A -85,B 0,C 180,E1 -14157.659,E2 -14157.659} C_VEL
LIN {X 0,Y 342.017,Z 496.743,A -85,B 0,C 180,E1 -14161.6,E2 -14161.6} C_VEL
LIN {X 0,Y 342.851,Z 490.478,A -85,B 0,C 180,E1 -14165.027,E2 -14165.027} C_VEL
LIN {X 0,Y 342.969,Z 487.101,A -85,B 0,C 180,E1 -14166.949,E2 -14166.949} C_VEL
LIN {X 0,Y 342.036,Z 481.174,A -85,B 0,C 180,E1 -14170.513,E2 -14170.513} C_VEL
LIN {X 0,Y 340.906,Z 474.871,A -85,B 0,C 180,E1 -14174.502,E2 -14174.502} C_VEL
LIN {X 0,Y 340.806,Z 474.034,A -85,B 0,C 180,E1 -14175.11,E2 -14175.11} C_VEL
LIN {X 0,Y 340.726,Z 474.045,A -85,B 0,C 180,E1 -14178.696,E2 -14178.696} C_VEL
LIN {X 0,Y 340.735,Z 474.039,A -85,B 0,C 180,E1 -14181.773,E2 -14181.773} C_VEL
LIN {X 0,Y 340.723,Z 474.04,A -85,B 0,C 180,E1 -14185.595,E2 -14185.595} C_VEL
LIN {X 0,Y 340.698,Z 474.046,A -85,B 0,C 180,E1 -14188.955,E2 -14188.955} C_VEL
LIN {X 0,Y 340.804,Z 474.033,A -85,B 0,C 180,E1 -14193.02,E2 -14193.02} C_VEL
LIN {X 0,Y 340.757,Z 474.036,A -85,B 0,C 180,E1 -14195.639,E2 -14195.639} C_VEL
LIN {X 0,Y 340.754,Z 474.037,A -85,B 0,C 180,E1 -14199.475,E2 -14199.475} C_VEL
LIN {X 0,Y 340.859,Z 474.024,A -85,B 0,C 180,E1 -14201.984,E2 -14201.984} C_VEL
LIN {X 0,Y 340.87,Z 474.022,A -85,B 0,C 180,E1 -14205.705,E2 -14205.705} C_VEL
LIN {X 0,Y 340.872,Z 474.022,A -85,B 0,C 180,E1 -14209.306,E2 -14209.306} C_VEL
LIN {X 0,Y 341.078,Z 473.999,A -85,B 0,C 180,E1 -14212.898,E2 -14212.898} C_VEL
LIN {X 0,Y 341.17,Z 473.984,A -85,B 0,C 180,E1 -14217.639,E2 -14217.639} C_VEL
LIN {X 0,Y 341.298,Z 473.97,A -85,B 0,C 180,E1 -14220,E2 -14220} C_VEL
LIN {X 0,Y 341.171,Z 473.989,A -85,B 0,C 180,E1 -14222.361,E2 -14222.361} C_VEL
LIN {X 0,Y 341.078,Z 473.997,A -85,B 0,C 180,E1 -14227.102,E2 -14227.102} C_VEL
LIN {X 0,Y 340.873,Z 474.025,A -85,B 0,C 180,E1 -14230.694,E2 -14230.694} C_VEL
LIN {X 0,Y 340.865,Z 474.028,A -85,B 0,C 180,E1 -14234.325,E2 -14234.325} C_VEL
LIN {X 0,Y 340.84,Z 474.031,A -85,B 0,C 180,E1 -14238.467,E2 -14238.467} C_VEL
LIN {X 0,Y 340.755,Z 474.038,A -85,B 0,C 180,E1 -14241.857,E2 -14241.857} C_VEL
LIN {X 0,Y 340.775,Z 474.034,A -85,B 0,C 180,E1 -14245.665,E2 -14245.665} C_VEL
LIN {X 0,Y 340.743,Z 474.043,A -85,B 0,C 180,E1 -14248.32,E2 -14248.32} C_VEL
LIN {X 0,Y 340.706,Z 474.043,A -85,B 0,C 180,E1 -14251.044,E2 -14251.044} C_VEL
LIN {X 0,Y 340.72,Z 474.04,A -85,B 0,C 180,E1 -14255.279,E2 -14255.279} C_VEL
LIN {X 0,Y 340.712,Z 474.047,A -85,B 0,C 180,E1 -14258.386,E2 -14258.386} C_VEL
LIN {X 0,Y 340.701,Z 474.047,A -85,B 0,C 180,E1 -14262.046,E2 -14262.046} C_VEL
LIN {X 0,Y 340.655,Z 474.054,A -85,B 0,C 180,E1 -14266.227,E2 -14266.227} C_VEL
LIN {X 0,Y 340.691,Z 474.046,A -85,B 0,C 180,E1 -14269.753,E2 -14269.753} C_VEL
LIN {X 0,Y 340.71,Z 474.042,A -85,B 0,C 180,E1 -14273.259,E2 -14273.259} C_VEL
LIN {X 0,Y 340.697,Z 474.049,A -85,B 0,C 180,E1 -14276.154,E2 -14276.154} C_VEL
LIN {X 0,Y 340.744,Z 474.042,A -85,B 0,C 180,E1 -14280.33,E2 -14280.33} C_VEL
LIN {X 0,Y 340.807,Z 474.03,A -85,B 0,C 180,E1 -14283.02,E2 -14283.02} C_VEL
LIN {X 0,Y 340.76,Z 474.037,A -85,B 0,C 180,E1 -14285.639,E2 -14285.639} C_VEL
LIN {X 0,Y 340.752,Z 474.037,A -85,B 0,C 180,E1 -14289.475,E2 -14289.475} C_VEL
LIN {X 0,Y 340.862,Z 474.028,A -85,B 0,C 180,E1 -14291.985,E2 -14291.985} C_VEL
LIN {X 0,Y 340.873,Z 474.024,A -85,B 0,C 180,E1 -14295.705,E2 -14295.705} C_VEL
LIN {X 0,Y 340.875,Z 474.022,A -85,B 0,C 180,E1 -14299.306,E2 -14299.306} C_VEL
LIN {X 0,Y 341.022,Z 474.003,A -85,B 0,C 180,E1 -14302.897,E2 -14302.897} C_VEL
LIN {X 0,Y 341.172,Z 473.987,A -85,B 0,C 180,E1 -14307.639,E2 -14307.639} C_VEL
LIN {X 0,Y 341.299,Z 473.974,A -85,B 0,C 180,E1 -14310,E2 -14310} C_VEL
LIN {X 0,Y 341.172,Z 473.987,A -85,B 0,C 180,E1 -14312.361,E2 -14312.361} C_VEL
LIN {X 0,Y 341.061,Z 473.998,A -85,B 0,C 180,E1 -14317.102,E2 -14317.102} C_VEL
LIN {X 0,Y 340.875,Z 474.022,A -85,B 0,C 180,E1 -14320.694,E2 -14320.694} C_VEL
LIN {X 0,Y 340.867,Z 474.024,A -85,B 0,C 180,E1 -14324.325,E2 -14324.325} C_VEL
LIN {X 0,Y 340.842,Z 474.027,A -85,B 0,C 180,E1 -14328.467,E2 -14328.467} C_VEL
LIN {X 0,Y 340.758,Z 474.041,A -85,B 0,C 180,E1 -14331.857,E2 -14331.857} C_VEL
LIN {X 0,Y 340.776,Z 474.038,A -85,B 0,C 180,E1 -14335.664,E2 -14335.664} C_VEL
LIN {X 0,Y 340.732,Z 474.041,A -85,B 0,C 180,E1 -14338.321,E2 -14338.321} C_VEL
LIN {X 0,Y 340.702,Z 474.043,A -85,B 0,C 180,E1 -14341.045,E2 -14341.045} C_VEL
LIN {X 0,Y 340.722,Z 474.042,A -85,B 0,C 180,E1 -14345.279,E2 -14345.279} C_VEL
LIN {X 0,Y 340.714,Z 474.042,A -85,B 0,C 180,E1 -14348.386,E2 -14348.386} C_VEL
LIN {X 0,Y 340.702,Z 474.046,A -85,B 0,C 180,E1 -14352.045,E2 -14352.045} C_VEL
LIN {X 0,Y 340.655,Z 474.05,A -85,B 0,C 180,E1 -14356.227,E2 -14356.227} C_VEL
LIN {X 0,Y 340.692,Z 474.05,A -85,B 0,C 180,E1 -14359.753,E2 -14359.753} C_VEL
LIN {X 0,Y 340.729,Z 474.045,A -85,B 0,C 180,E1 -14361.772,E2 -14361.772} C_VEL
LIN {X 0,Y 340.557,Z 474.061,A -85,B 0,C 180,E1 -14364.701,E2 -14364.701} C_VEL
LIN {X 0,Y 340.27,Z 474.101,A -85,B 0,C 180,E1 -14367.868,E2 -14367.868} C_VEL
LIN {X 0,Y 339.9,Z 474.149,A -85,B 0,C 180,E1 -14371.604,E2 -14371.604} C_VEL
LIN {X 0,Y 339.735,Z 474.169,A -85,B 0,C 180,E1 -14372.928,E2 -14372.928} C_VEL
LIN {X 0,Y 339.632,Z 475.612,A -85,B 0,C 180,E1 -14374.642,E2 -14374.642} C_VEL
LIN {X 0,Y 338.933,Z 476.589,A -85,B 0,C 180,E1 -14375.617,E2 -14375.617} C_VEL
LIN {X 0,Y 336.031,Z 478.347,A -85,B 0,C 180,E1 -14377.198,E2 -14377.198} C_VEL
LIN {X 0,Y 333.581,Z 479.78,A -85,B 0,C 180,E1 -14378.477,E2 -14378.477} C_VEL
LIN {X 0,Y 332.523,Z 480.821,A -85,B 0,C 180,E1 -14379.47,E2 -14379.47} C_VEL
LIN {X 0,Y 332.434,Z 481.153,A -85,B 0,C 180,E1 -14379.807,E2 -14379.807} C_VEL
LIN {X 0,Y 332.436,Z 481.572,A -85,B 0,C 180,E1 -14380.169,E2 -14380.169} C_VEL
LIN {X 0,Y 335.097,Z 494.658,A -85,B 0,C 180,E1 -14380.927,E2 -14380.927} C_VEL
LIN {X 0,Y 337.873,Z 508.431,A -85,B 0,C 180,E1 -14381.976,E2 -14381.976} C_VEL
LIN {X 0,Y 337.773,Z 513.978,A -85,B 0,C 180,E1 -14382.44,E2 -14382.44} C_VEL
LIN {X 0,Y 336.84,Z 526.032,A -85,B 0,C 180,E1 -14383.623,E2 -14383.623} C_VEL
LIN {X 0,Y 335.893,Z 537.276,A -85,B 0,C 180,E1 -14384.993,E2 -14384.993} C_VEL
LIN {X 0,Y 335.059,Z 546.401,A -85,B 0,C 180,E1 -14386.351,E2 -14386.351} C_VEL
LIN {X 0,Y 334.142,Z 556.36,A -85,B 0,C 180,E1 -14388.166,E2 -14388.166} C_VEL
LIN {X 0,Y 333.442,Z 564.457,A -85,B 0,C 180,E1 -14389.986,E2 -14389.986} C_VEL
LIN {X 0,Y 332.844,Z 571.907,A -85,B 0,C 180,E1 -14392.111,E2 -14392.111} C_VEL
LIN {X 0,Y 332.53,Z 576.927,A -85,B 0,C 180,E1 -14393.934,E2 -14393.934} C_VEL
LIN {X 0,Y 332.337,Z 580.807,A -85,B 0,C 180,E1 -14395.755,E2 -14395.755} C_VEL
LIN {X 0,Y 332.239,Z 583.634,A -85,B 0,C 180,E1 -14397.575,E2 -14397.575} C_VEL
LIN {X 0,Y 332.236,Z 584.997,A -85,B 0,C 180,E1 -14398.788,E2 -14398.788} C_VEL
LIN {X 0,Y 332.254,Z 585.906,A -85,B 0,C 180,E1 -14400,E2 -14400} C_VEL
LIN {X 0,Y 332.345,Z 586.41,A -85,B 0,C 180,E1 -14401.212,E2 -14401.212} C_VEL
LIN {X 0,Y 332.486,Z 586.524,A -85,B 0,C 180,E1 -14402.423,E2 -14402.423} C_VEL
LIN {X 0,Y 332.697,Z 586.235,A -85,B 0,C 180,E1 -14403.633,E2 -14403.633} C_VEL
LIN {X 0,Y 332.894,Z 585.508,A -85,B 0,C 180,E1 -14404.844,E2 -14404.844} C_VEL
LIN {X 0,Y 332.953,Z 584.407,A -85,B 0,C 180,E1 -14406.058,E2 -14406.058} C_VEL
LIN {X 0,Y 333.8,Z 581.284,A -85,B 0,C 180,E1 -14408.283,E2 -14408.283} C_VEL
LIN {X 0,Y 334.692,Z 577.189,A -85,B 0,C 180,E1 -14410.281,E2 -14410.281} C_VEL
LIN {X 0,Y 335.85,Z 572.313,A -85,B 0,C 180,E1 -14412.079,E2 -14412.079} C_VEL
LIN {X 0,Y 337.402,Z 565.109,A -85,B 0,C 180,E1 -14414.167,E2 -14414.167} C_VEL
LIN {X 0,Y 338.97,Z 557.478,A -85,B 0,C 180,E1 -14415.945,E2 -14415.945} C_VEL
LIN {X 0,Y 341.128,Z 547.931,A -85,B 0,C 180,E1 -14417.691,E2 -14417.691} C_VEL
LIN {X 0,Y 343.236,Z 536.757,A -85,B 0,C 180,E1 -14419.36,E2 -14419.36} C_VEL
LIN {X 0,Y 345.308,Z 525.395,A -85,B 0,C 180,E1 -14420.709,E2 -14420.709} C_VEL
LIN {X 0,Y 345.966,Z 521.241,A -85,B 0,C 180,E1 -14421.135,E2 -14421.135} C_VEL
LIN {X 0,Y 344.93,Z 515.631,A -85,B 0,C 180,E1 -14421.899,E2 -14421.899} C_VEL
LIN {X 0,Y 341.766,Z 505.879,A -85,B 0,C 180,E1 -14423.327,E2 -14423.327} C_VEL
LIN {X 0,Y 337.274,Z 495.928,A -85,B 0,C 180,E1 -14424.884,E2 -14424.884} C_VEL
LIN {X 0,Y 336.18,Z 493.627,A -85,B 0,C 180,E1 -14425.24,E2 -14425.24} C_VEL
LIN {X 0,Y 334.996,Z 492.012,A -85,B 0,C 180,E1 -14425.562,E2 -14425.562} C_VEL
LIN {X 0,Y 334.152,Z 489.559,A -85,B 0,C 180,E1 -14425.926,E2 -14425.926} C_VEL
LIN {X 0,Y 334.544,Z 488.549,A -85,B 0,C 180,E1 -14428.893,E2 -14428.893} C_VEL
LIN {X 0,Y 334.925,Z 487.891,A -85,B 0,C 180,E1 -14431.641,E2 -14431.641} C_VEL
LIN {X 0,Y 335.473,Z 487.492,A -85,B 0,C 180,E1 -14435.211,E2 -14435.211} C_VEL
LIN {X 0,Y 335.849,Z 487.752,A -85,B 0,C 180,E1 -14438.887,E2 -14438.887} C_VEL
LIN {X 0,Y 336.031,Z 488.565,A -85,B 0,C 180,E1 -14442.011,E2 -14442.011} C_VEL
LIN {X 0,Y 336.349,Z 490.004,A -85,B 0,C 180,E1 -14445.27,E2 -14445.27} C_VEL
LIN {X 0,Y 336.714,Z 492.245,A -85,B 0,C 180,E1 -14448.712,E2 -14448.712} C_VEL
LIN {X 0,Y 336.958,Z 494.422,A -85,B 0,C 180,E1 -14451.265,E2 -14451.265} C_VEL
LIN {X 0,Y 336.994,Z 495.928,A -85,B 0,C 180,E1 -14452.786,E2 -14452.786} C_VEL
LIN {X 0,Y 336.365,Z 499.293,A -85,B 0,C 180,E1 -14455.657,E2 -14455.657} C_VEL
LIN {X 0,Y 335.339,Z 504.182,A -85,B 0,C 180,E1 -14459.235,E2 -14459.235} C_VEL
LIN {X 0,Y 334.284,Z 510.215,A -85,B 0,C 180,E1 -14463.127,E2 -14463.127} C_VEL
LIN {X 0,Y 334.101,Z 511.665,A -85,B 0,C 180,E1 -14464.01,E2 -14464.01} C_VEL
LIN {X 0,Y 335.072,Z 515.334,A -85,B 0,C 180,E1 -14464.41,E2 -14464.41} C_VEL
LIN {X 0,Y 337.099,Z 521.37,A -85,B 0,C 180,E1 -14465.146,E2 -14465.146} C_VEL
LIN {X 0,Y 340.373,Z 534.852,A -85,B 0,C 180,E1 -14466.68,E2 -14466.68} C_VEL
LIN {X 0,Y 341.88,Z 546.682,A -85,B 0,C 180,E1 -14467.999,E2 -14467.999} C_VEL
LIN {X 0,Y 342.069,Z 555.736,A -85,B 0,C 180,E1 -14469.027,E2 -14469.027} C_VEL
LIN {X 0,Y 341.393,Z 565.029,A -85,B 0,C 180,E1 -14470.143,E2 -14470.143} C_VEL
LIN {X 0,Y 339.341,Z 576.077,A -85,B 0,C 180,E1 -14471.588,E2 -14471.588} C_VEL
LIN {X 0,Y 337.59,Z 585.3,A -85,B 0,C 180,E1 -14473.055,E2 -14473.055} C_VEL
LIN {X 0,Y 336.026,Z 593.099,A -85,B 0,C 180,E1 -14474.534,E2 -14474.534} C_VEL
LIN {X 0,Y 334.741,Z 600.992,A -85,B 0,C 180,E1 -14476.338,E2 -14476.338} C_VEL
LIN {X 0,Y 333.402,Z 608.436,A -85,B 0,C 180,E1 -14478.448,E2 -14478.448} C_VEL
LIN {X 0,Y 332.748,Z 613.53,A -85,B 0,C 180,E1 -14480.272,E2 -14480.272} C_VEL
LIN {X 0,Y 332.32,Z 617.549,A -85,B 0,C 180,E1 -14482.099,E2 -14482.099} C_VEL
LIN {X 0,Y 332.094,Z 620.755,A -85,B 0,C 180,E1 -14484.069,E2 -14484.069} C_VEL
LIN {X 0,Y 332.059,Z 623.107,A -85,B 0,C 180,E1 -14486.359,E2 -14486.359} C_VEL
LIN {X 0,Y 332.081,Z 623.722,A -85,B 0,C 180,E1 -14487.574,E2 -14487.574} C_VEL
LIN {X 0,Y 332.252,Z 623.927,A -85,B 0,C 180,E1 -14488.788,E2 -14488.788} C_VEL
LIN {X 0,Y 332.278,Z 623.712,A -85,B 0,C 180,E1 -14490,E2 -14490} C_VEL
LIN {X 0,Y 332.293,Z 623.079,A -85,B 0,C 180,E1 -14491.212,E2 -14491.212} C_VEL
LIN {X 0,Y 332.215,Z 621.963,A -85,B 0,C 180,E1 -14492.425,E2 -14492.425} C_VEL
LIN {X 0,Y 332.118,Z 620.409,A -85,B 0,C 180,E1 -14493.64,E2 -14493.64} C_VEL
LIN {X 0,Y 332.24,Z 618.435,A -85,B 0,C 180,E1 -14494.854,E2 -14494.854} C_VEL
LIN {X 0,Y 332.265,Z 614.639,A -85,B 0,C 180,E1 -14496.619,E2 -14496.619} C_VEL
LIN {X 0,Y 332.506,Z 608.358,A -85,B 0,C 180,E1 -14498.815,E2 -14498.815} C_VEL
LIN {X 0,Y 332.9,Z 601.629,A -85,B 0,C 180,E1 -14500.645,E2 -14500.645} C_VEL
LIN {X 0,Y 333.644,Z 593.309,A -85,B 0,C 180,E1 -14502.469,E2 -14502.469} C_VEL
LIN {X 0,Y 334.38,Z 584.777,A -85,B 0,C 180,E1 -14503.987,E2 -14503.987} C_VEL
LIN {X 0,Y 335.188,Z 575.82,A -85,B 0,C 180,E1 -14505.313,E2 -14505.313} C_VEL
LIN {X 0,Y 336.226,Z 564.358,A -85,B 0,C 180,E1 -14506.703,E2 -14506.703} C_VEL
LIN {X 0,Y 336.795,Z 556.851,A -85,B 0,C 180,E1 -14507.456,E2 -14507.456} C_VEL
LIN {X 0,Y 335.583,Z 544.143,A -85,B 0,C 180,E1 -14508.558,E2 -14508.558} C_VEL
LIN {X 0,Y 334.063,Z 530.631,A -85,B 0,C 180,E1 -14509.466,E2 -14509.466} C_VEL
LIN {X 0,Y 332.787,Z 518.788,A -85,B 0,C 180,E1 -14510.07,E2 -14510.07} C_VEL
LIN {X 0,Y 333.403,Z 510.908,A -85,B 0,C 180,E1 -14514.271,E2 -14514.271} C_VEL
LIN {X 0,Y 334.162,Z 504.08,A -85,B 0,C 180,E1 -14517.953,E2 -14517.953} C_VEL
LIN {X 0,Y 334.969,Z 497.382,A -85,B 0,C 180,E1 -14521.636,E2 -14521.636} C_VEL
LIN {X 0,Y 335.844,Z 490.87,A -85,B 0,C 180,E1 -14525.301,E2 -14525.301} C_VEL
LIN {X 0,Y 335.843,Z 487.343,A -85,B 0,C 180,E1 -14527.363,E2 -14527.363} C_VEL
LIN {X 0,Y 334.905,Z 481.546,A -85,B 0,C 180,E1 -14530.934,E2 -14530.934} C_VEL
LIN {X 0,Y 333.817,Z 475.186,A -85,B 0,C 180,E1 -14535.07,E2 -14535.07} C_VEL
LIN {X 0,Y 333.727,Z 474.916,A -85,B 0,C 180,E1 -14535.726,E2 -14535.726} C_VEL
LIN {X 0,Y 333.702,Z 474.916,A -85,B 0,C 180,E1 -14539.304,E2 -14539.304} C_VEL
LIN {X 0,Y 333.665,Z 474.921,A -85,B 0,C 180,E1 -14543.168,E2 -14543.168} C_VEL
LIN {X 0,Y 333.675,Z 474.919,A -85,B 0,C 180,E1 -14545.341,E2 -14545.341} C_VEL
LIN {X 0,Y 333.691,Z 474.916,A -85,B 0,C 180,E1 -14549.637,E2 -14549.637} C_VEL
LIN {X 0,Y 333.74,Z 474.913,A -85,B 0,C 180,E1 -14552.401,E2 -14552.401} C_VEL
LIN {X 0,Y 333.728,Z 474.913,A -85,B 0,C 180,E1 -14555.091,E2 -14555.091} C_VEL
LIN {X 0,Y 333.686,Z 474.919,A -85,B 0,C 180,E1 -14559.02,E2 -14559.02} C_VEL
LIN {X 0,Y 333.794,Z 474.903,A -85,B 0,C 180,E1 -14561.59,E2 -14561.59} C_VEL
LIN {X 0,Y 333.809,Z 474.901,A -85,B 0,C 180,E1 -14565.577,E2 -14565.577} C_VEL
LIN {X 0,Y 333.835,Z 474.899,A -85,B 0,C 180,E1 -14569.078,E2 -14569.078} C_VEL
LIN {X 0,Y 334.027,Z 474.878,A -85,B 0,C 180,E1 -14572.748,E2 -14572.748} C_VEL
LIN {X 0,Y 333.811,Z 474.902,A -85,B 0,C 180,E1 -14575.169,E2 -14575.169} C_VEL
LIN {X 0,Y 334.107,Z 474.864,A -85,B 0,C 180,E1 -14577.589,E2 -14577.589} C_VEL
LIN {X 0,Y 334.249,Z 474.848,A -85,B 0,C 180,E1 -14580,E2 -14580} C_VEL
LIN {X 0,Y 334.108,Z 474.869,A -85,B 0,C 180,E1 -14582.411,E2 -14582.411} C_VEL
LIN {X 0,Y 334.027,Z 474.874,A -85,B 0,C 180,E1 -14587.253,E2 -14587.253} C_VEL
LIN {X 0,Y 333.836,Z 474.899,A -85,B 0,C 180,E1 -14590.922,E2 -14590.922} C_VEL
LIN {X 0,Y 333.81,Z 474.905,A -85,B 0,C 180,E1 -14594.634,E2 -14594.634} C_VEL
LIN {X 0,Y 333.799,Z 474.906,A -85,B 0,C 180,E1 -14598.656,E2 -14598.656} C_VEL
LIN {X 0,Y 333.694,Z 474.921,A -85,B 0,C 180,E1 -14602.278,E2 -14602.278} C_VEL
LIN {X 0,Y 333.738,Z 474.915,A -85,B 0,C 180,E1 -14606.246,E2 -14606.246} C_VEL
LIN {X 0,Y 333.713,Z 474.914,A -85,B 0,C 180,E1 -14608.972,E2 -14608.972} C_VEL
LIN {X 0,Y 333.648,Z 474.924,A -85,B 0,C 180,E1 -14612.588,E2 -14612.588} C_VEL
LIN {X 0,Y 333.679,Z 474.922,A -85,B 0,C 180,E1 -14616.139,E2 -14616.139} C_VEL
LIN {X 0,Y 333.649,Z 474.921,A -85,B 0,C 180,E1 -14619.193,E2 -14619.193} C_VEL
LIN {X 0,Y 333.635,Z 474.927,A -85,B 0,C 180,E1 -14622.5,E2 -14622.5} C_VEL
LIN {X 0,Y 333.599,Z 474.931,A -85,B 0,C 180,E1 -14625.955,E2 -14625.955} C_VEL
LIN {X 0,Y 333.65,Z 474.921,A -85,B 0,C 180,E1 -14629.316,E2 -14629.316} C_VEL
LIN {X 0,Y 333.67,Z 474.919,A -85,B 0,C 180,E1 -14633.168,E2 -14633.168} C_VEL
LIN {X 0,Y 333.642,Z 474.923,A -85,B 0,C 180,E1 -14636.792,E2 -14636.792} C_VEL
LIN {X 0,Y 333.697,Z 474.917,A -85,B 0,C 180,E1 -14639.713,E2 -14639.713} C_VEL
LIN {X 0,Y 333.743,Z 474.913,A -85,B 0,C 180,E1 -14642.401,E2 -14642.401} C_VEL
LIN {X 0,Y 333.73,Z 474.911,A -85,B 0,C 180,E1 -14645.091,E2 -14645.091} C_VEL
LIN {X 0,Y 333.685,Z 474.917,A -85,B 0,C 180,E1 -14649.02,E2 -14649.02} C_VEL
LIN {X 0,Y 333.798,Z 474.904,A -85,B 0,C 180,E1 -14651.59,E2 -14651.59} C_VEL
LIN {X 0,Y 333.812,Z 474.902,A -85,B 0,C 180,E1 -14655.577,E2 -14655.577} C_VEL
LIN {X 0,Y 333.838,Z 474.898,A -85,B 0,C 180,E1 -14659.078,E2 -14659.078} C_VEL
LIN {X 0,Y 333.974,Z 474.881,A -85,B 0,C 180,E1 -14662.747,E2 -14662.747} C_VEL
LIN {X 0,Y 333.808,Z 474.901,A -85,B 0,C 180,E1 -14665.169,E2 -14665.169} C_VEL
LIN {X 0,Y 334.109,Z 474.866,A -85,B 0,C 180,E1 -14667.589,E2 -14667.589} C_VEL
LIN {X 0,Y 334.25,Z 474.852,A -85,B 0,C 180,E1 -14670,E2 -14670} C_VEL
LIN {X 0,Y 334.11,Z 474.866,A -85,B 0,C 180,E1 -14672.411,E2 -14672.411} C_VEL
LIN {X 0,Y 334.017,Z 474.881,A -85,B 0,C 180,E1 -14676.039,E2 -14676.039} C_VEL
LIN {X 0,Y 333.963,Z 474.883,A -85,B 0,C 180,E1 -14678.471,E2 -14678.471} C_VEL
LIN {X 0,Y 333.796,Z 474.907,A -85,B 0,C 180,E1 -14682.155,E2 -14682.155} C_VEL
LIN {X 0,Y 333.782,Z 474.91,A -85,B 0,C 180,E1 -14685.886,E2 -14685.886} C_VEL
LIN {X 0,Y 333.801,Z 474.903,A -85,B 0,C 180,E1 -14688.656,E2 -14688.656} C_VEL
LIN {X 0,Y 333.696,Z 474.917,A -85,B 0,C 180,E1 -14692.278,E2 -14692.278} C_VEL
LIN {X 0,Y 333.739,Z 474.912,A -85,B 0,C 180,E1 -14696.246,E2 -14696.246} C_VEL
LIN {X 0,Y 333.694,Z 474.916,A -85,B 0,C 180,E1 -14698.974,E2 -14698.974} C_VEL
LIN {X 0,Y 333.649,Z 474.921,A -85,B 0,C 180,E1 -14702.588,E2 -14702.588} C_VEL
LIN {X 0,Y 333.68,Z 474.92,A -85,B 0,C 180,E1 -14706.139,E2 -14706.139} C_VEL
LIN {X 0,Y 333.65,Z 474.922,A -85,B 0,C 180,E1 -14709.192,E2 -14709.192} C_VEL
LIN {X 0,Y 333.636,Z 474.923,A -85,B 0,C 180,E1 -14712.5,E2 -14712.5} C_VEL
LIN {X 0,Y 333.6,Z 474.931,A -85,B 0,C 180,E1 -14715.955,E2 -14715.955} C_VEL
LIN {X 0,Y 333.651,Z 474.923,A -85,B 0,C 180,E1 -14719.315,E2 -14719.315} C_VEL
LIN {X 0,Y 333.635,Z 474.924,A -85,B 0,C 180,E1 -14723.175,E2 -14723.175} C_VEL
LIN {X 0,Y 333.306,Z 474.964,A -85,B 0,C 180,E1 -14726.754,E2 -14726.754} C_VEL
LIN {X 0,Y 333.011,Z 475.005,A -85,B 0,C 180,E1 -14729.915,E2 -14729.915} C_VEL
LIN {X 0,Y 332.736,Z 475.043,A -85,B 0,C 180,E1 -14732.514,E2 -14732.514} C_VEL
LIN {X 0,Y 332.594,Z 475.365,A -85,B 0,C 180,E1 -14733.656,E2 -14733.656} C_VEL
LIN {X 0,Y 332.496,Z 477.839,A -85,B 0,C 180,E1 -14736.321,E2 -14736.321} C_VEL
LIN {X 0,Y 332.434,Z 481.153,A -85,B 0,C 180,E1 -14739.807,E2 -14739.807} C_VEL
LIN {X 0,Y 332.43,Z 482.094,A -85,B 0,C 180,E1 -14740.066,E2 -14740.066} C_VEL
LIN {X 0,Y 332.428,Z 484.489,A -85,B 0,C 180,E1 -14740.281,E2 -14740.281} C_VEL
LIN {X 0,Y 332.102,Z 495.635,A -85,B 0,C 180,E1 -14740.878,E2 -14740.878} C_VEL
LIN {X 0,Y 330.847,Z 506.37,A -85,B 0,C 180,E1 -14741.539,E2 -14741.539} C_VEL
LIN {X 0,Y 330.971,Z 510.257,A -85,B 0,C 180,E1 -14741.895,E2 -14741.895} C_VEL
LIN {X 0,Y 330.187,Z 521.987,A -85,B 0,C 180,E1 -14742.979,E2 -14742.979} C_VEL
LIN {X 0,Y 329.224,Z 533.992,A -85,B 0,C 180,E1 -14744.365,E2 -14744.365} C_VEL
LIN {X 0,Y 328.334,Z 543.712,A -85,B 0,C 180,E1 -14745.749,E2 -14745.749} C_VEL
LIN {X 0,Y 327.276,Z 554.337,A -85,B 0,C 180,E1 -14747.599,E2 -14747.599} C_VEL
LIN {X 0,Y 326.533,Z 562.857,A -85,B 0,C 180,E1 -14749.458,E2 -14749.458} C_VEL
LIN {X 0,Y 325.925,Z 569.769,A -85,B 0,C 180,E1 -14751.318,E2 -14751.318} C_VEL
LIN {X 0,Y 325.575,Z 575.388,A -85,B 0,C 180,E1 -14753.207,E2 -14753.207} C_VEL
LIN {X 0,Y 325.348,Z 579.68,A -85,B 0,C 180,E1 -14755.043,E2 -14755.043} C_VEL
LIN {X 0,Y 325.206,Z 581.983,A -85,B 0,C 180,E1 -14756.283,E2 -14756.283} C_VEL
LIN {X 0,Y 325.144,Z 583.82,A -85,B 0,C 180,E1 -14757.522,E2 -14757.522} C_VEL
LIN {X 0,Y 325.141,Z 585.25,A -85,B 0,C 180,E1 -14758.761,E2 -14758.761} C_VEL
LIN {X 0,Y 325.178,Z 586.269,A -85,B 0,C 180,E1 -14760,E2 -14760} C_VEL
LIN {X 0,Y 325.269,Z 586.835,A -85,B 0,C 180,E1 -14761.238,E2 -14761.238} C_VEL
LIN {X 0,Y 325.418,Z 587.008,A -85,B 0,C 180,E1 -14762.475,E2 -14762.475} C_VEL
LIN {X 0,Y 325.639,Z 586.788,A -85,B 0,C 180,E1 -14763.712,E2 -14763.712} C_VEL
LIN {X 0,Y 325.843,Z 586.172,A -85,B 0,C 180,E1 -14764.949,E2 -14764.949} C_VEL
LIN {X 0,Y 325.926,Z 585.146,A -85,B 0,C 180,E1 -14766.189,E2 -14766.189} C_VEL
LIN {X 0,Y 326.837,Z 582.172,A -85,B 0,C 180,E1 -14768.449,E2 -14768.449} C_VEL
LIN {X 0,Y 327.792,Z 578.214,A -85,B 0,C 180,E1 -14770.5,E2 -14770.5} C_VEL
LIN {X 0,Y 329.014,Z 573.535,A -85,B 0,C 180,E1 -14772.334,E2 -14772.334} C_VEL
LIN {X 0,Y 330.686,Z 566.565,A -85,B 0,C 180,E1 -14774.461,E2 -14774.461} C_VEL
LIN {X 0,Y 332.323,Z 559.123,A -85,B 0,C 180,E1 -14776.273,E2 -14776.273} C_VEL
LIN {X 0,Y 334.611,Z 549.978,A -85,B 0,C 180,E1 -14778.047,E2 -14778.047} C_VEL
LIN {X 0,Y 336.934,Z 538.775,A -85,B 0,C 180,E1 -14779.813,E2 -14779.813} C_VEL
LIN {X 0,Y 339.204,Z 527.06,A -85,B 0,C 180,E1 -14781.258,E2 -14781.258} C_VEL
LIN {X 0,Y 339.925,Z 523.068,A -85,B 0,C 180,E1 -14781.689,E2 -14781.689} C_VEL
LIN {X 0,Y 338.166,Z 515.104,A -85,B 0,C 180,E1 -14782.894,E2 -14782.894} C_VEL
LIN {X 0,Y 334.356,Z 504.753,A -85,B 0,C 180,E1 -14784.569,E2 -14784.569} C_VEL
LIN {X 0,Y 331.525,Z 498.526,A -85,B 0,C 180,E1 -14785.63,E2 -14785.63} C_VEL
LIN {X 0,Y 329.427,Z 494.654,A -85,B 0,C 180,E1 -14786.358,E2 -14786.358} C_VEL
LIN {X 0,Y 328.236,Z 493.087,A -85,B 0,C 180,E1 -14786.721,E2 -14786.721} C_VEL
LIN {X 0,Y 327.328,Z 490.496,A -85,B 0,C 180,E1 -14787.146,E2 -14787.146} C_VEL
LIN {X 0,Y 327.886,Z 489.48,A -85,B 0,C 180,E1 -14790.977,E2 -14790.977} C_VEL
LIN {X 0,Y 328.28,Z 489.083,A -85,B 0,C 180,E1 -14793.822,E2 -14793.822} C_VEL
LIN {X 0,Y 328.707,Z 489.056,A -85,B 0,C 180,E1 -14796.774,E2 -14796.774} C_VEL
LIN {X 0,Y 328.974,Z 489.509,A -85,B 0,C 180,E1 -14799.859,E2 -14799.859} C_VEL
LIN {X 0,Y 329.269,Z 490.718,A -85,B 0,C 180,E1 -14803.472,E2 -14803.472} C_VEL
LIN {X 0,Y 329.609,Z 492.599,A -85,B 0,C 180,E1 -14806.975,E2 -14806.975} C_VEL
LIN {X 0,Y 329.946,Z 495.064,A -85,B 0,C 180,E1 -14810.281,E2 -14810.281} C_VEL
LIN {X 0,Y 330.035,Z 496.62,A -85,B 0,C 180,E1 -14811.99,E2 -14811.99} C_VEL
LIN {X 0,Y 329.777,Z 498.824,A -85,B 0,C 180,E1 -14814.08,E2 -14814.08} C_VEL
LIN {X 0,Y 329.178,Z 501.591,A -85,B 0,C 180,E1 -14816.373,E2 -14816.373} C_VEL
LIN {X 0,Y 328.14,Z 506.258,A -85,B 0,C 180,E1 -14819.78,E2 -14819.78} C_VEL
LIN {X 0,Y 327.352,Z 510.858,A -85,B 0,C 180,E1 -14822.813,E2 -14822.813} C_VEL
LIN {X 0,Y 328.244,Z 514.343,A -85,B 0,C 180,E1 -14823.224,E2 -14823.224} C_VEL
LIN {X 0,Y 328.989,Z 515.755,A -85,B 0,C 180,E1 -14823.458,E2 -14823.458} C_VEL
LIN {X 0,Y 332.47,Z 527.796,A -85,B 0,C 180,E1 -14824.99,E2 -14824.99} C_VEL
LIN {X 0,Y 334.888,Z 540.214,A -85,B 0,C 180,E1 -14826.501,E2 -14826.501} C_VEL
LIN {X 0,Y 335.829,Z 551.568,A -85,B 0,C 180,E1 -14827.871,E2 -14827.871} C_VEL
LIN {X 0,Y 335.307,Z 563.173,A -85,B 0,C 180,E1 -14829.286,E2 -14829.286} C_VEL
LIN {X 0,Y 333.32,Z 574.223,A -85,B 0,C 180,E1 -14830.764,E2 -14830.764} C_VEL
LIN {X 0,Y 331.174,Z 584.448,A -85,B 0,C 180,E1 -14832.398,E2 -14832.398} C_VEL
LIN {X 0,Y 329.215,Z 593.728,A -85,B 0,C 180,E1 -14834.206,E2 -14834.206} C_VEL
LIN {X 0,Y 327.648,Z 602.48,A -85,B 0,C 180,E1 -14836.352,E2 -14836.352} C_VEL
LIN {X 0,Y 326.419,Z 608.605,A -85,B 0,C 180,E1 -14838.197,E2 -14838.197} C_VEL
LIN {X 0,Y 325.736,Z 613.554,A -85,B 0,C 180,E1 -14840.06,E2 -14840.06} C_VEL
LIN {X 0,Y 325.251,Z 617.445,A -85,B 0,C 180,E1 -14841.926,E2 -14841.926} C_VEL
LIN {X 0,Y 324.999,Z 620.769,A -85,B 0,C 180,E1 -14844.12,E2 -14844.12} C_VEL
LIN {X 0,Y 324.982,Z 622.739,A -85,B 0,C 180,E1 -14846.28,E2 -14846.28} C_VEL
LIN {X 0,Y 325.17,Z 623.45,A -85,B 0,C 180,E1 -14848.761,E2 -14848.761} C_VEL
LIN {X 0,Y 325.219,Z 623.189,A -85,B 0,C 180,E1 -14850,E2 -14850} C_VEL
LIN {X 0,Y 325.233,Z 622.466,A -85,B 0,C 180,E1 -14851.238,E2 -14851.238} C_VEL
LIN {X 0,Y 325.128,Z 621.293,A -85,B 0,C 180,E1 -14852.478,E2 -14852.478} C_VEL
LIN {X 0,Y 325.103,Z 618.707,A -85,B 0,C 180,E1 -14854.339,E2 -14854.339} C_VEL
LIN {X 0,Y 325.193,Z 615.044,A -85,B 0,C 180,E1 -14856.203,E2 -14856.203} C_VEL
LIN {X 0,Y 325.325,Z 610.201,A -85,B 0,C 180,E1 -14858.072,E2 -14858.072} C_VEL
LIN {X 0,Y 325.673,Z 604.069,A -85,B 0,C 180,E1 -14859.941,E2 -14859.941} C_VEL
LIN {X 0,Y 326.241,Z 596.429,A -85,B 0,C 180,E1 -14861.809,E2 -14861.809} C_VEL
LIN {X 0,Y 327.037,Z 586.887,A -85,B 0,C 180,E1 -14863.673,E2 -14863.673} C_VEL
LIN {X 0,Y 328.026,Z 576.594,A -85,B 0,C 180,E1 -14865.298,E2 -14865.298} C_VEL
LIN {X 0,Y 329.139,Z 565.053,A -85,B 0,C 180,E1 -14866.754,E2 -14866.754} C_VEL
LIN {X 0,Y 329.697,Z 556.114,A -85,B 0,C 180,E1 -14867.684,E2 -14867.684} C_VEL
LIN {X 0,Y 328.545,Z 544.569,A -85,B 0,C 180,E1 -14868.715,E2 -14868.715} C_VEL
LIN {X 0,Y 327.103,Z 531.455,A -85,B 0,C 180,E1 -14869.643,E2 -14869.643} C_VEL
LIN {X 0,Y 325.736,Z 518.403,A -85,B 0,C 180,E1 -14870.359,E2 -14870.359} C_VEL
LIN {X 0,Y 326.388,Z 510.415,A -85,B 0,C 180,E1 -14874.733,E2 -14874.733} C_VEL
LIN {X 0,Y 327.276,Z 502.936,A -85,B 0,C 180,E1 -14878.892,E2 -14878.892} C_VEL
LIN {X 0,Y 328.027,Z 496.761,A -85,B 0,C 180,E1 -14882.386,E2 -14882.386} C_VEL
LIN {X 0,Y 328.776,Z 491.779,A -85,B 0,C 180,E1 -14885.251,E2 -14885.251} C_VEL
LIN {X 0,Y 328.877,Z 489.246,A -85,B 0,C 180,E1 -14886.752,E2 -14886.752} C_VEL
LIN {X 0,Y 328.152,Z 484.076,A -85,B 0,C 180,E1 -14889.979,E2 -14889.979} C_VEL
LIN {X 0,Y 327.194,Z 478.783,A -85,B 0,C 180,E1 -14893.42,E2 -14893.42} C_VEL
LIN {X 0,Y 326.707,Z 475.791,A -85,B 0,C 180,E1 -14895.531,E2 -14895.531} C_VEL
LIN {X 0,Y 326.635,Z 475.795,A -85,B 0,C 180,E1 -14899.798,E2 -14899.798} C_VEL
LIN {X 0,Y 326.631,Z 475.799,A -85,B 0,C 180,E1 -14902.953,E2 -14902.953} C_VEL
LIN {X 0,Y 326.607,Z 475.799,A -85,B 0,C 180,E1 -14905.981,E2 -14905.981} C_VEL
LIN {X 0,Y 326.648,Z 475.796,A -85,B 0,C 180,E1 -14910.34,E2 -14910.34} C_VEL
LIN {X 0,Y 326.691,Z 475.792,A -85,B 0,C 180,E1 -14914.516,E2 -14914.516} C_VEL
LIN {X 0,Y 326.649,Z 475.798,A -85,B 0,C 180,E1 -14918.546,E2 -14918.546} C_VEL
LIN {X 0,Y 326.745,Z 475.782,A -85,B 0,C 180,E1 -14921.178,E2 -14921.178} C_VEL
LIN {X 0,Y 326.764,Z 475.779,A -85,B 0,C 180,E1 -14925.433,E2 -14925.433} C_VEL
LIN {X 0,Y 326.771,Z 475.781,A -85,B 0,C 180,E1 -14928.839,E2 -14928.839} C_VEL
LIN {X 0,Y 326.981,Z 475.757,A -85,B 0,C 180,E1 -14932.591,E2 -14932.591} C_VEL
LIN {X 0,Y 326.779,Z 475.778,A -85,B 0,C 180,E1 -14935.065,E2 -14935.065} C_VEL
LIN {X 0,Y 327.048,Z 475.743,A -85,B 0,C 180,E1 -14937.537,E2 -14937.537} C_VEL
LIN {X 0,Y 327.201,Z 475.726,A -85,B 0,C 180,E1 -14940,E2 -14940} C_VEL
LIN {X 0,Y 327.049,Z 475.749,A -85,B 0,C 180,E1 -14942.463,E2 -14942.463} C_VEL
LIN {X 0,Y 326.973,Z 475.752,A -85,B 0,C 180,E1 -14946.665,E2 -14946.665} C_VEL
LIN {X 0,Y 326.816,Z 475.774,A -85,B 0,C 180,E1 -14949.906,E2 -14949.906} C_VEL
LIN {X 0,Y 326.761,Z 475.779,A -85,B 0,C 180,E1 -14953.686,E2 -14953.686} C_VEL
LIN {X 0,Y 326.701,Z 475.787,A -85,B 0,C 180,E1 -14957.528,E2 -14957.528} C_VEL
LIN {X 0,Y 326.667,Z 475.794,A -85,B 0,C 180,E1 -14960.135,E2 -14960.135} C_VEL
LIN {X 0,Y 326.654,Z 475.796,A -85,B 0,C 180,E1 -14964.129,E2 -14964.129} C_VEL
LIN {X 0,Y 326.687,Z 475.79,A -85,B 0,C 180,E1 -14966.858,E2 -14966.858} C_VEL
LIN {X 0,Y 326.641,Z 475.797,A -85,B 0,C 180,E1 -14970.611,E2 -14970.611} C_VEL
LIN {X 0,Y 326.61,Z 475.801,A -85,B 0,C 180,E1 -14974.02,E2 -14974.02} C_VEL
LIN {X 0,Y 326.63,Z 475.795,A -85,B 0,C 180,E1 -14977.239,E2 -14977.239} C_VEL
LIN {X 0,Y 326.58,Z 475.802,A -85,B 0,C 180,E1 -14981.132,E2 -14981.132} C_VEL
LIN {X 0,Y 326.53,Z 475.809,A -85,B 0,C 180,E1 -14984.743,E2 -14984.743} C_VEL
LIN {X 0,Y 326.579,Z 475.807,A -85,B 0,C 180,E1 -14988.155,E2 -14988.155} C_VEL
LIN {X 0,Y 326.627,Z 475.796,A -85,B 0,C 180,E1 -14991.392,E2 -14991.392} C_VEL
LIN {X 0,Y 326.623,Z 475.797,A -85,B 0,C 180,E1 -14994.851,E2 -14994.851} C_VEL
LIN {X 0,Y 326.613,Z 475.798,A -85,B 0,C 180,E1 -14997.456,E2 -14997.456} C_VEL
LIN {X 0,Y 326.651,Z 475.797,A -85,B 0,C 180,E1 -15000.34,E2 -15000.34} C_VEL
LIN {X 0,Y 326.693,Z 475.79,A -85,B 0,C 180,E1 -15004.517,E2 -15004.517} C_VEL
LIN {X 0,Y 326.65,Z 475.795,A -85,B 0,C 180,E1 -15008.546,E2 -15008.546} C_VEL
LIN {X 0,Y 326.748,Z 475.781,A -85,B 0,C 180,E1 -15011.178,E2 -15011.178} C_VEL
LIN {X 0,Y 326.767,Z 475.779,A -85,B 0,C 180,E1 -15015.433,E2 -15015.433} C_VEL
LIN {X 0,Y 326.774,Z 475.778,A -85,B 0,C 180,E1 -15018.839,E2 -15018.839} C_VEL
LIN {X 0,Y 326.928,Z 475.759,A -85,B 0,C 180,E1 -15022.589,E2 -15022.589} C_VEL
LIN {X 0,Y 326.775,Z 475.777,A -85,B 0,C 180,E1 -15025.065,E2 -15025.065} C_VEL
LIN {X 0,Y 327.05,Z 475.745,A -85,B 0,C 180,E1 -15027.537,E2 -15027.537} C_VEL
LIN {X 0,Y 327.202,Z 475.73,A -85,B 0,C 180,E1 -15030,E2 -15030} C_VEL
LIN {X 0,Y 327.05,Z 475.745,A -85,B 0,C 180,E1 -15032.463,E2 -15032.463} C_VEL
LIN {X 0,Y 326.992,Z 475.754,A -85,B 0,C 180,E1 -15036.169,E2 -15036.169} C_VEL
LIN {X 0,Y 326.81,Z 475.779,A -85,B 0,C 180,E1 -15039.907,E2 -15039.907} C_VEL
LIN {X 0,Y 326.763,Z 475.782,A -85,B 0,C 180,E1 -15043.685,E2 -15043.685} C_VEL
LIN {X 0,Y 326.704,Z 475.788,A -85,B 0,C 180,E1 -15047.528,E2 -15047.528} C_VEL
LIN {X 0,Y 326.669,Z 475.794,A -85,B 0,C 180,E1 -15050.135,E2 -15050.135} C_VEL
LIN {X 0,Y 326.656,Z 475.795,A -85,B 0,C 180,E1 -15054.129,E2 -15054.129} C_VEL
LIN {X 0,Y 326.687,Z 475.788,A -85,B 0,C 180,E1 -15056.858,E2 -15056.858} C_VEL
LIN {X 0,Y 326.638,Z 475.795,A -85,B 0,C 180,E1 -15060.61,E2 -15060.61} C_VEL
LIN {X 0,Y 326.611,Z 475.801,A -85,B 0,C 180,E1 -15064.019,E2 -15064.019} C_VEL
LIN {X 0,Y 326.631,Z 475.796,A -85,B 0,C 180,E1 -15067.239,E2 -15067.239} C_VEL
LIN {X 0,Y 326.581,Z 475.802,A -85,B 0,C 180,E1 -15071.131,E2 -15071.131} C_VEL
LIN {X 0,Y 326.531,Z 475.808,A -85,B 0,C 180,E1 -15074.743,E2 -15074.743} C_VEL
LIN {X 0,Y 326.579,Z 475.804,A -85,B 0,C 180,E1 -15078.154,E2 -15078.154} C_VEL
LIN {X 0,Y 326.596,Z 475.802,A -85,B 0,C 180,E1 -15081.387,E2 -15081.387} C_VEL
LIN {X 0,Y 326.46,Z 475.817,A -85,B 0,C 180,E1 -15084.461,E2 -15084.461} C_VEL
LIN {X 0,Y 326.226,Z 475.849,A -85,B 0,C 180,E1 -15087.412,E2 -15087.412} C_VEL
LIN {X 0,Y 325.922,Z 475.885,A -85,B 0,C 180,E1 -15090.267,E2 -15090.267} C_VEL
LIN {X 0,Y 325.593,Z 475.93,A -85,B 0,C 180,E1 -15093.045,E2 -15093.045} C_VEL
LIN {X 0,Y 325.512,Z 477.335,A -85,B 0,C 180,E1 -15095.068,E2 -15095.068} C_VEL
LIN {X 0,Y 325.385,Z 480.483,A -85,B 0,C 180,E1 -15098.458,E2 -15098.458} C_VEL
LIN {X 0,Y 325.377,Z 481.972,A -85,B 0,C 180,E1 -15099.911,E2 -15099.911} C_VEL
LIN {X 0,Y 328.071,Z 495.496,A -85,B 0,C 180,E1 -15100.721,E2 -15100.721} C_VEL
LIN {X 0,Y 330.864,Z 509.436,A -85,B 0,C 180,E1 -15101.821,E2 -15101.821} C_VEL
LIN {X 0,Y 330.971,Z 510.257,A -85,B 0,C 180,E1 -15101.895,E2 -15101.895} C_VEL
LIN {X 0,Y 330.676,Z 513.226,A -85,B 0,C 180,E1 -15102.142,E2 -15102.142} C_VEL
LIN {X 0,Y 328.739,Z 517.167,A -85,B 0,C 180,E1 -15102.441,E2 -15102.441} C_VEL
LIN {X 0,Y 323.699,Z 524.572,A -85,B 0,C 180,E1 -15103.048,E2 -15103.048} C_VEL
LIN {X 0,Y 322.727,Z 527.902,A -85,B 0,C 180,E1 -15103.407,E2 -15103.407} C_VEL
LIN {X 0,Y 321.743,Z 538.676,A -85,B 0,C 180,E1 -15104.804,E2 -15104.804} C_VEL
LIN {X 0,Y 320.821,Z 548.556,A -85,B 0,C 180,E1 -15106.379,E2 -15106.379} C_VEL
LIN {X 0,Y 319.908,Z 558.288,A -85,B 0,C 180,E1 -15108.275,E2 -15108.275} C_VEL
LIN {X 0,Y 319.18,Z 566.122,A -85,B 0,C 180,E1 -15110.174,E2 -15110.174} C_VEL
LIN {X 0,Y 318.643,Z 573.429,A -85,B 0,C 180,E1 -15112.395,E2 -15112.395} C_VEL
LIN {X 0,Y 318.323,Z 578.321,A -85,B 0,C 180,E1 -15114.298,E2 -15114.298} C_VEL
LIN {X 0,Y 318.135,Z 582.088,A -85,B 0,C 180,E1 -15116.2,E2 -15116.2} C_VEL
LIN {X 0,Y 318.054,Z 584.005,A -85,B 0,C 180,E1 -15117.467,E2 -15117.467} C_VEL
LIN {X 0,Y 318.046,Z 585.499,A -85,B 0,C 180,E1 -15118.734,E2 -15118.734} C_VEL
LIN {X 0,Y 318.085,Z 586.588,A -85,B 0,C 180,E1 -15120,E2 -15120} C_VEL
LIN {X 0,Y 318.197,Z 587.26,A -85,B 0,C 180,E1 -15121.265,E2 -15121.265} C_VEL
LIN {X 0,Y 318.584,Z 587.346,A -85,B 0,C 180,E1 -15123.794,E2 -15123.794} C_VEL
LIN {X 0,Y 318.797,Z 586.817,A -85,B 0,C 180,E1 -15125.059,E2 -15125.059} C_VEL
LIN {X 0,Y 318.903,Z 585.893,A -85,B 0,C 180,E1 -15126.326,E2 -15126.326} C_VEL
LIN {X 0,Y 319.99,Z 582.728,A -85,B 0,C 180,E1 -15128.844,E2 -15128.844} C_VEL
LIN {X 0,Y 320.911,Z 579.279,A -85,B 0,C 180,E1 -15130.728,E2 -15130.728} C_VEL
LIN {X 0,Y 322.186,Z 574.761,A -85,B 0,C 180,E1 -15132.599,E2 -15132.599} C_VEL
LIN {X 0,Y 323.668,Z 569.092,A -85,B 0,C 180,E1 -15134.46,E2 -15134.46} C_VEL
LIN {X 0,Y 325.413,Z 562.21,A -85,B 0,C 180,E1 -15136.306,E2 -15136.306} C_VEL
LIN {X 0,Y 327.675,Z 553.649,A -85,B 0,C 180,E1 -15138.119,E2 -15138.119} C_VEL
LIN {X 0,Y 330.165,Z 543.222,A -85,B 0,C 180,E1 -15139.912,E2 -15139.912} C_VEL
LIN {X 0,Y 332.584,Z 532.001,A -85,B 0,C 180,E1 -15141.464,E2 -15141.464} C_VEL
LIN {X 0,Y 333.917,Z 525.161,A -85,B 0,C 180,E1 -15142.262,E2 -15142.262} C_VEL
LIN {X 0,Y 332.332,Z 517.991,A -85,B 0,C 180,E1 -15143.426,E2 -15143.426} C_VEL
LIN {X 0,Y 329.047,Z 508.536,A -85,B 0,C 180,E1 -15145.066,E2 -15145.066} C_VEL
LIN {X 0,Y 325.75,Z 501.465,A -85,B 0,C 180,E1 -15146.426,E2 -15146.426} C_VEL
LIN {X 0,Y 322.806,Z 495.718,A -85,B 0,C 180,E1 -15147.595,E2 -15147.595} C_VEL
LIN {X 0,Y 321.641,Z 494.276,A -85,B 0,C 180,E1 -15147.99,E2 -15147.99} C_VEL
LIN {X 0,Y 320.582,Z 491.526,A -85,B 0,C 180,E1 -15148.478,E2 -15148.478} C_VEL
LIN {X 0,Y 321.036,Z 490.825,A -85,B 0,C 180,E1 -15151.695,E2 -15151.695} C_VEL
LIN {X 0,Y 321.467,Z 490.554,A -85,B 0,C 180,E1 -15154.64,E2 -15154.64} C_VEL
LIN {X 0,Y 321.887,Z 490.679,A -85,B 0,C 180,E1 -15157.687,E2 -15157.687} C_VEL
LIN {X 0,Y 322.108,Z 491.359,A -85,B 0,C 180,E1 -15160.886,E2 -15160.886} C_VEL
LIN {X 0,Y 322.396,Z 492.643,A -85,B 0,C 180,E1 -15164.233,E2 -15164.233} C_VEL
LIN {X 0,Y 322.722,Z 494.53,A -85,B 0,C 180,E1 -15167.538,E2 -15167.538} C_VEL
LIN {X 0,Y 323.031,Z 497.097,A -85,B 0,C 180,E1 -15170.88,E2 -15170.88} C_VEL
LIN {X 0,Y 322.892,Z 499.792,A -85,B 0,C 180,E1 -15173.643,E2 -15173.643} C_VEL
LIN {X 0,Y 321.976,Z 503.697,A -85,B 0,C 180,E1 -15176.928,E2 -15176.928} C_VEL
LIN {X 0,Y 320.91,Z 508.531,A -85,B 0,C 180,E1 -15180.478,E2 -15180.478} C_VEL
LIN {X 0,Y 320.685,Z 509.952,A -85,B 0,C 180,E1 -15181.451,E2 -15181.451} C_VEL
LIN {X 0,Y 321.642,Z 513.642,A -85,B 0,C 180,E1 -15181.95,E2 -15181.95} C_VEL
LIN {X 0,Y 322.748,Z 516.603,A -85,B 0,C 180,E1 -15182.424,E2 -15182.424} C_VEL
LIN {X 0,Y 325.626,Z 525.791,A -85,B 0,C 180,E1 -15183.74,E2 -15183.74} C_VEL
LIN {X 0,Y 328.109,Z 536.879,A -85,B 0,C 180,E1 -15185.225,E2 -15185.225} C_VEL
LIN {X 0,Y 329.469,Z 548.512,A -85,B 0,C 180,E1 -15186.729,E2 -15186.729} C_VEL
LIN {X 0,Y 329.549,Z 557.797,A -85,B 0,C 180,E1 -15187.922,E2 -15187.922} C_VEL
LIN {X 0,Y 328.318,Z 568.242,A -85,B 0,C 180,E1 -15189.317,E2 -15189.317} C_VEL
LIN {X 0,Y 326.07,Z 578.413,A -85,B 0,C 180,E1 -15190.81,E2 -15190.81} C_VEL
LIN {X 0,Y 324.165,Z 586.987,A -85,B 0,C 180,E1 -15192.33,E2 -15192.33} C_VEL
LIN {X 0,Y 322.149,Z 595.736,A -85,B 0,C 180,E1 -15194.189,E2 -15194.189} C_VEL
LIN {X 0,Y 320.767,Z 602.887,A -85,B 0,C 180,E1 -15196.054,E2 -15196.054} C_VEL
LIN {X 0,Y 319.456,Z 608.804,A -85,B 0,C 180,E1 -15197.936,E2 -15197.936} C_VEL
LIN {X 0,Y 318.519,Z 614.944,A -85,B 0,C 180,E1 -15200.474,E2 -15200.474} C_VEL
LIN {X 0,Y 318.074,Z 618.364,A -85,B 0,C 180,E1 -15202.382,E2 -15202.382} C_VEL
LIN {X 0,Y 317.893,Z 620.726,A -85,B 0,C 180,E1 -15204.19,E2 -15204.19} C_VEL
LIN {X 0,Y 317.906,Z 622.365,A -85,B 0,C 180,E1 -15206.197,E2 -15206.197} C_VEL
LIN {X 0,Y 318.091,Z 622.971,A -85,B 0,C 180,E1 -15208.734,E2 -15208.734} C_VEL
LIN {X 0,Y 318.161,Z 622.625,A -85,B 0,C 180,E1 -15210,E2 -15210} C_VEL
LIN {X 0,Y 318.173,Z 621.833,A -85,B 0,C 180,E1 -15211.266,E2 -15211.266} C_VEL
LIN {X 0,Y 318.043,Z 620.604,A -85,B 0,C 180,E1 -15212.533,E2 -15212.533} C_VEL
LIN {X 0,Y 318.047,Z 617.911,A -85,B 0,C 180,E1 -15214.436,E2 -15214.436} C_VEL
LIN {X 0,Y 318.122,Z 614.134,A -85,B 0,C 180,E1 -15216.342,E2 -15216.342} C_VEL
LIN {X 0,Y 318.261,Z 609.175,A -85,B 0,C 180,E1 -15218.252,E2 -15218.252} C_VEL
LIN {X 0,Y 318.615,Z 602.91,A -85,B 0,C 180,E1 -15220.164,E2 -15220.164} C_VEL
LIN {X 0,Y 319.268,Z 595.057,A -85,B 0,C 180,E1 -15222.071,E2 -15222.071} C_VEL
LIN {X 0,Y 320.104,Z 585.339,A -85,B 0,C 180,E1 -15223.976,E2 -15223.976} C_VEL
LIN {X 0,Y 321.003,Z 576.078,A -85,B 0,C 180,E1 -15225.447,E2 -15225.447} C_VEL
LIN {X 0,Y 322.153,Z 564.302,A -85,B 0,C 180,E1 -15226.965,E2 -15226.965} C_VEL
LIN {X 0,Y 322.66,Z 556.958,A -85,B 0,C 180,E1 -15227.754,E2 -15227.754} C_VEL
LIN {X 0,Y 321.352,Z 543.593,A -85,B 0,C 180,E1 -15228.985,E2 -15228.985} C_VEL
LIN {X 0,Y 319.937,Z 530.492,A -85,B 0,C 180,E1 -15229.92,E2 -15229.92} C_VEL
LIN {X 0,Y 318.653,Z 518.065,A -85,B 0,C 180,E1 -15230.622,E2 -15230.622} C_VEL
LIN {X 0,Y 319.304,Z 510.788,A -85,B 0,C 180,E1 -15234.721,E2 -15234.721} C_VEL
LIN {X 0,Y 320.19,Z 503.493,A -85,B 0,C 180,E1 -15238.874,E2 -15238.874} C_VEL
LIN {X 0,Y 321.182,Z 496.115,A -85,B 0,C 180,E1 -15243.164,E2 -15243.164} C_VEL
LIN {X 0,Y 321.787,Z 491.13,A -85,B 0,C 180,E1 -15246.135,E2 -15246.135} C_VEL
LIN {X 0,Y 321.603,Z 487.937,A -85,B 0,C 180,E1 -15248.121,E2 -15248.121} C_VEL
LIN {X 0,Y 320.818,Z 483.348,A -85,B 0,C 180,E1 -15251.086,E2 -15251.086} C_VEL
LIN {X 0,Y 319.751,Z 477.155,A -85,B 0,C 180,E1 -15255.304,E2 -15255.304} C_VEL
LIN {X 0,Y 319.654,Z 476.669,A -85,B 0,C 180,E1 -15255.796,E2 -15255.796} C_VEL
LIN {X 0,Y 319.581,Z 476.679,A -85,B 0,C 180,E1 -15258.72,E2 -15258.72} C_VEL
LIN {X 0,Y 319.582,Z 476.676,A -85,B 0,C 180,E1 -15262.343,E2 -15262.343} C_VEL
LIN {X 0,Y 319.561,Z 476.678,A -85,B 0,C 180,E1 -15265.124,E2 -15265.124} C_VEL
LIN {X 0,Y 319.567,Z 476.677,A -85,B 0,C 180,E1 -15269.059,E2 -15269.059} C_VEL
LIN {X 0,Y 319.607,Z 476.674,A -85,B 0,C 180,E1 -15272.498,E2 -15272.498} C_VEL
LIN {X 0,Y 319.606,Z 476.671,A -85,B 0,C 180,E1 -15275.304,E2 -15275.304} C_VEL
LIN {X 0,Y 319.598,Z 476.672,A -85,B 0,C 180,E1 -15278.048,E2 -15278.048} C_VEL
LIN {X 0,Y 319.69,Z 476.662,A -85,B 0,C 180,E1 -15280.962,E2 -15280.962} C_VEL
LIN {X 0,Y 319.732,Z 476.655,A -85,B 0,C 180,E1 -15285.276,E2 -15285.276} C_VEL
LIN {X 0,Y 319.759,Z 476.652,A -85,B 0,C 180,E1 -15289.873,E2 -15289.873} C_VEL
LIN {X 0,Y 319.935,Z 476.634,A -85,B 0,C 180,E1 -15292.426,E2 -15292.426} C_VEL
LIN {X 0,Y 319.748,Z 476.654,A -85,B 0,C 180,E1 -15294.956,E2 -15294.956} C_VEL
LIN {X 0,Y 319.991,Z 476.622,A -85,B 0,C 180,E1 -15297.483,E2 -15297.483} C_VEL
LIN {X 0,Y 320.153,Z 476.604,A -85,B 0,C 180,E1 -15300,E2 -15300} C_VEL
LIN {X 0,Y 319.993,Z 476.628,A -85,B 0,C 180,E1 -15302.518,E2 -15302.518} C_VEL
LIN {X 0,Y 319.933,Z 476.631,A -85,B 0,C 180,E1 -15306.655,E2 -15306.655} C_VEL
LIN {X 0,Y 319.76,Z 476.654,A -85,B 0,C 180,E1 -15310.127,E2 -15310.127} C_VEL
LIN {X 0,Y 319.733,Z 476.657,A -85,B 0,C 180,E1 -15314.725,E2 -15314.725} C_VEL
LIN {X 0,Y 319.691,Z 476.66,A -85,B 0,C 180,E1 -15319.038,E2 -15319.038} C_VEL
LIN {X 0,Y 319.572,Z 476.674,A -85,B 0,C 180,E1 -15323.32,E2 -15323.32} C_VEL
LIN {X 0,Y 319.637,Z 476.67,A -85,B 0,C 180,E1 -15326.088,E2 -15326.088} C_VEL
LIN {X 0,Y 319.591,Z 476.673,A -85,B 0,C 180,E1 -15328.934,E2 -15328.934} C_VEL
LIN {X 0,Y 319.535,Z 476.681,A -85,B 0,C 180,E1 -15331.862,E2 -15331.862} C_VEL
LIN {X 0,Y 319.582,Z 476.674,A -85,B 0,C 180,E1 -15335.543,E2 -15335.543} C_VEL
LIN {X 0,Y 319.575,Z 476.677,A -85,B 0,C 180,E1 -15338.008,E2 -15338.008} C_VEL
LIN {X 0,Y 319.528,Z 476.681,A -85,B 0,C 180,E1 -15341.597,E2 -15341.597} C_VEL
LIN {X 0,Y 319.491,Z 476.685,A -85,B 0,C 180,E1 -15345.258,E2 -15345.258} C_VEL
LIN {X 0,Y 319.531,Z 476.681,A -85,B 0,C 180,E1 -15348.712,E2 -15348.712} C_VEL
LIN {X 0,Y 319.581,Z 476.678,A -85,B 0,C 180,E1 -15352.344,E2 -15352.344} C_VEL
LIN {X 0,Y 319.563,Z 476.676,A -85,B 0,C 180,E1 -15355.124,E2 -15355.124} C_VEL
LIN {X 0,Y 319.569,Z 476.675,A -85,B 0,C 180,E1 -15359.059,E2 -15359.059} C_VEL
LIN {X 0,Y 319.609,Z 476.673,A -85,B 0,C 180,E1 -15362.498,E2 -15362.498} C_VEL
LIN {X 0,Y 319.608,Z 476.67,A -85,B 0,C 180,E1 -15365.304,E2 -15365.304} C_VEL
LIN {X 0,Y 319.6,Z 476.676,A -85,B 0,C 180,E1 -15368.048,E2 -15368.048} C_VEL
LIN {X 0,Y 319.693,Z 476.66,A -85,B 0,C 180,E1 -15370.962,E2 -15370.962} C_VEL
LIN {X 0,Y 319.735,Z 476.654,A -85,B 0,C 180,E1 -15375.276,E2 -15375.276} C_VEL
LIN {X 0,Y 319.756,Z 476.656,A -85,B 0,C 180,E1 -15379.873,E2 -15379.873} C_VEL
LIN {X 0,Y 319.915,Z 476.634,A -85,B 0,C 180,E1 -15383.694,E2 -15383.694} C_VEL
LIN {X 0,Y 319.993,Z 476.623,A -85,B 0,C 180,E1 -15387.483,E2 -15387.483} C_VEL
LIN {X 0,Y 320.154,Z 476.608,A -85,B 0,C 180,E1 -15390,E2 -15390} C_VEL
LIN {X 0,Y 319.994,Z 476.623,A -85,B 0,C 180,E1 -15392.518,E2 -15392.518} C_VEL
LIN {X 0,Y 319.946,Z 476.63,A -85,B 0,C 180,E1 -15396.306,E2 -15396.306} C_VEL
LIN {X 0,Y 319.841,Z 476.641,A -85,B 0,C 180,E1 -15398.848,E2 -15398.848} C_VEL
LIN {X 0,Y 319.686,Z 476.66,A -85,B 0,C 180,E1 -15402.7,E2 -15402.7} C_VEL
LIN {X 0,Y 319.704,Z 476.659,A -85,B 0,C 180,E1 -15405.296,E2 -15405.296} C_VEL
LIN {X 0,Y 319.679,Z 476.662,A -85,B 0,C 180,E1 -15409.255,E2 -15409.255} C_VEL
LIN {X 0,Y 319.574,Z 476.675,A -85,B 0,C 180,E1 -15413.319,E2 -15413.319} C_VEL
LIN {X 0,Y 319.638,Z 476.67,A -85,B 0,C 180,E1 -15416.088,E2 -15416.088} C_VEL
LIN {X 0,Y 319.583,Z 476.673,A -85,B 0,C 180,E1 -15418.934,E2 -15418.934} C_VEL
LIN {X 0,Y 319.535,Z 476.685,A -85,B 0,C 180,E1 -15421.862,E2 -15421.862} C_VEL
LIN {X 0,Y 319.584,Z 476.676,A -85,B 0,C 180,E1 -15425.543,E2 -15425.543} C_VEL
LIN {X 0,Y 319.577,Z 476.677,A -85,B 0,C 180,E1 -15428.008,E2 -15428.008} C_VEL
LIN {X 0,Y 319.529,Z 476.684,A -85,B 0,C 180,E1 -15431.597,E2 -15431.597} C_VEL
LIN {X 0,Y 319.492,Z 476.686,A -85,B 0,C 180,E1 -15435.257,E2 -15435.257} C_VEL
LIN {X 0,Y 319.531,Z 476.679,A -85,B 0,C 180,E1 -15438.712,E2 -15438.712} C_VEL
LIN {X 0,Y 319.539,Z 476.679,A -85,B 0,C 180,E1 -15442.354,E2 -15442.354} C_VEL
LIN {X 0,Y 319.359,Z 476.702,A -85,B 0,C 180,E1 -15445.098,E2 -15445.098} C_VEL
LIN {X 0,Y 318.987,Z 476.749,A -85,B 0,C 180,E1 -15449.234,E2 -15449.234} C_VEL
LIN {X 0,Y 318.664,Z 476.797,A -85,B 0,C 180,E1 -15452.409,E2 -15452.409} C_VEL
LIN {X 0,Y 318.455,Z 476.861,A -85,B 0,C 180,E1 -15453.808,E2 -15453.808} C_VEL
LIN {X 0,Y 318.324,Z 479.386,A -85,B 0,C 180,E1 -15456.583,E2 -15456.583} C_VEL
LIN {X 0,Y 318.307,Z 482.302,A -85,B 0,C 180,E1 -15459.65,E2 -15459.65} C_VEL
LIN {X 0,Y 320.781,Z 494.892,A -85,B 0,C 180,E1 -15460.406,E2 -15460.406} C_VEL
LIN {X 0,Y 323.397,Z 508.311,A -85,B 0,C 180,E1 -15461.468,E2 -15461.468} C_VEL
LIN {X 0,Y 323.979,Z 512.282,A -85,B 0,C 180,E1 -15461.83,E2 -15461.83} C_VEL
LIN {X 0,Y 323.035,Z 524.197,A -85,B 0,C 180,E1 -15462.985,E2 -15462.985} C_VEL
LIN {X 0,Y 322.727,Z 527.902,A -85,B 0,C 180,E1 -15463.407,E2 -15463.407} C_VEL
LIN {X 0,Y 321.788,Z 532.765,A -85,B 0,C 180,E1 -15463.979,E2 -15463.979} C_VEL
LIN {X 0,Y 318.265,Z 540.338,A -85,B 0,C 180,E1 -15464.94,E2 -15464.94} C_VEL
LIN {X 0,Y 314.599,Z 547.435,A -85,B 0,C 180,E1 -15466.021,E2 -15466.021} C_VEL
LIN {X 0,Y 313.462,Z 551.563,A -85,B 0,C 180,E1 -15466.772,E2 -15466.772} C_VEL
LIN {X 0,Y 312.639,Z 560.517,A -85,B 0,C 180,E1 -15468.656,E2 -15468.656} C_VEL
LIN {X 0,Y 311.945,Z 568.055,A -85,B 0,C 180,E1 -15470.599,E2 -15470.599} C_VEL
LIN {X 0,Y 311.567,Z 573.204,A -85,B 0,C 180,E1 -15472.221,E2 -15472.221} C_VEL
LIN {X 0,Y 311.235,Z 578.244,A -85,B 0,C 180,E1 -15474.168,E2 -15474.168} C_VEL
LIN {X 0,Y 311.067,Z 582.131,A -85,B 0,C 180,E1 -15476.113,E2 -15476.113} C_VEL
LIN {X 0,Y 310.967,Z 584.166,A -85,B 0,C 180,E1 -15477.409,E2 -15477.409} C_VEL
LIN {X 0,Y 310.95,Z 585.724,A -85,B 0,C 180,E1 -15478.705,E2 -15478.705} C_VEL
LIN {X 0,Y 311.109,Z 587.644,A -85,B 0,C 180,E1 -15481.294,E2 -15481.294} C_VEL
LIN {X 0,Y 311.289,Z 587.989,A -85,B 0,C 180,E1 -15482.588,E2 -15482.588} C_VEL
LIN {X 0,Y 311.531,Z 587.903,A -85,B 0,C 180,E1 -15483.88,E2 -15483.88} C_VEL
LIN {X 0,Y 311.735,Z 587.441,A -85,B 0,C 180,E1 -15485.174,E2 -15485.174} C_VEL
LIN {X 0,Y 311.881,Z 586.622,A -85,B 0,C 180,E1 -15486.469,E2 -15486.469} C_VEL
LIN {X 0,Y 312.932,Z 583.997,A -85,B 0,C 180,E1 -15488.818,E2 -15488.818} C_VEL
LIN {X 0,Y 314.03,Z 580.356,A -85,B 0,C 180,E1 -15490.966,E2 -15490.966} C_VEL
LIN {X 0,Y 315.391,Z 576.013,A -85,B 0,C 180,E1 -15492.875,E2 -15492.875} C_VEL
LIN {X 0,Y 317.275,Z 569.582,A -85,B 0,C 180,E1 -15495.086,E2 -15495.086} C_VEL
LIN {X 0,Y 319.166,Z 562.672,A -85,B 0,C 180,E1 -15496.963,E2 -15496.963} C_VEL
LIN {X 0,Y 321.601,Z 554.173,A -85,B 0,C 180,E1 -15498.804,E2 -15498.804} C_VEL
LIN {X 0,Y 324.199,Z 544.131,A -85,B 0,C 180,E1 -15500.583,E2 -15500.583} C_VEL
LIN {X 0,Y 326.647,Z 533.552,A -85,B 0,C 180,E1 -15502.081,E2 -15502.081} C_VEL
LIN {X 0,Y 327.936,Z 527.379,A -85,B 0,C 180,E1 -15502.848,E2 -15502.848} C_VEL
LIN {X 0,Y 326.793,Z 521.684,A -85,B 0,C 180,E1 -15503.848,E2 -15503.848} C_VEL
LIN {X 0,Y 323.456,Z 511.483,A -85,B 0,C 180,E1 -15505.757,E2 -15505.757} C_VEL
LIN {X 0,Y 320.649,Z 505.214,A -85,B 0,C 180,E1 -15507.061,E2 -15507.061} C_VEL
LIN {X 0,Y 318.466,Z 500.863,A -85,B 0,C 180,E1 -15508.026,E2 -15508.026} C_VEL
LIN {X 0,Y 317.004,Z 498.455,A -85,B 0,C 180,E1 -15508.634,E2 -15508.634} C_VEL
LIN {X 0,Y 316.582,Z 497.353,A -85,B 0,C 180,E1 -15508.857,E2 -15508.857} C_VEL
LIN {X 0,Y 314.91,Z 495.397,A -85,B 0,C 180,E1 -15509.496,E2 -15509.496} C_VEL
LIN {X 0,Y 313.837,Z 492.6,A -85,B 0,C 180,E1 -15510.102,E2 -15510.102} C_VEL
LIN {X 0,Y 314.18,Z 492.237,A -85,B 0,C 180,E1 -15512.47,E2 -15512.47} C_VEL
LIN {X 0,Y 314.652,Z 492.096,A -85,B 0,C 180,E1 -15515.502,E2 -15515.502} C_VEL
LIN {X 0,Y 315.034,Z 492.406,A -85,B 0,C 180,E1 -15518.665,E2 -15518.665} C_VEL
LIN {X 0,Y 315.284,Z 493.305,A -85,B 0,C 180,E1 -15521.969,E2 -15521.969} C_VEL
LIN {X 0,Y 315.593,Z 494.856,A -85,B 0,C 180,E1 -15525.448,E2 -15525.448} C_VEL
LIN {X 0,Y 315.974,Z 497.215,A -85,B 0,C 180,E1 -15529.134,E2 -15529.134} C_VEL
LIN {X 0,Y 316.129,Z 499.145,A -85,B 0,C 180,E1 -15531.502,E2 -15531.502} C_VEL
LIN {X 0,Y 315.98,Z 500.785,A -85,B 0,C 180,E1 -15533.198,E2 -15533.198} C_VEL
LIN {X 0,Y 315.241,Z 504.1,A -85,B 0,C 180,E1 -15536.127,E2 -15536.127} C_VEL
LIN {X 0,Y 314.105,Z 508.93,A -85,B 0,C 180,E1 -15539.866,E2 -15539.866} C_VEL
LIN {X 0,Y 315.029,Z 512.662,A -85,B 0,C 180,E1 -15540.465,E2 -15540.465} C_VEL
LIN {X 0,Y 315.846,Z 514.287,A -85,B 0,C 180,E1 -15540.806,E2 -15540.806} C_VEL
LIN {X 0,Y 319.572,Z 526.458,A -85,B 0,C 180,E1 -15542.757,E2 -15542.757} C_VEL
LIN {X 0,Y 321.668,Z 535.525,A -85,B 0,C 180,E1 -15544.089,E2 -15544.089} C_VEL
LIN {X 0,Y 323.159,Z 546.281,A -85,B 0,C 180,E1 -15545.593,E2 -15545.593} C_VEL
LIN {X 0,Y 323.466,Z 557.505,A -85,B 0,C 180,E1 -15547.146,E2 -15547.146} C_VEL
LIN {X 0,Y 322.089,Z 568.869,A -85,B 0,C 180,E1 -15548.73,E2 -15548.73} C_VEL
LIN {X 0,Y 319.466,Z 579.648,A -85,B 0,C 180,E1 -15550.398,E2 -15550.398} C_VEL
LIN {X 0,Y 317.475,Z 587.943,A -85,B 0,C 180,E1 -15551.945,E2 -15551.945} C_VEL
LIN {X 0,Y 315.333,Z 596.478,A -85,B 0,C 180,E1 -15553.867,E2 -15553.867} C_VEL
LIN {X 0,Y 313.64,Z 604.277,A -85,B 0,C 180,E1 -15556.061,E2 -15556.061} C_VEL
LIN {X 0,Y 312.19,Z 610.682,A -85,B 0,C 180,E1 -15558.31,E2 -15558.31} C_VEL
LIN {X 0,Y 311.48,Z 614.965,A -85,B 0,C 180,E1 -15560.257,E2 -15560.257} C_VEL
LIN {X 0,Y 311.015,Z 618.243,A -85,B 0,C 180,E1 -15562.208,E2 -15562.208} C_VEL
LIN {X 0,Y 310.795,Z 620.676,A -85,B 0,C 180,E1 -15564.253,E2 -15564.253} C_VEL
LIN {X 0,Y 310.832,Z 621.996,A -85,B 0,C 180,E1 -15566.11,E2 -15566.11} C_VEL
LIN {X 0,Y 310.817,Z 622.439,A -85,B 0,C 180,E1 -15567.408,E2 -15567.408} C_VEL
LIN {X 0,Y 311.013,Z 622.458,A -85,B 0,C 180,E1 -15568.705,E2 -15568.705} C_VEL
LIN {X 0,Y 311.104,Z 622.032,A -85,B 0,C 180,E1 -15570,E2 -15570} C_VEL
LIN {X 0,Y 311.114,Z 621.183,A -85,B 0,C 180,E1 -15571.294,E2 -15571.294} C_VEL
LIN {X 0,Y 310.961,Z 619.897,A -85,B 0,C 180,E1 -15572.591,E2 -15572.591} C_VEL
LIN {X 0,Y 310.992,Z 617.095,A -85,B 0,C 180,E1 -15574.536,E2 -15574.536} C_VEL
LIN {X 0,Y 311.065,Z 613.201,A -85,B 0,C 180,E1 -15576.486,E2 -15576.486} C_VEL
LIN {X 0,Y 311.265,Z 607.1,A -85,B 0,C 180,E1 -15578.766,E2 -15578.766} C_VEL
LIN {X 0,Y 311.663,Z 600.406,A -85,B 0,C 180,E1 -15580.722,E2 -15580.722} C_VEL
LIN {X 0,Y 312.418,Z 592.134,A -85,B 0,C 180,E1 -15582.67,E2 -15582.67} C_VEL
LIN {X 0,Y 313.343,Z 581.762,A -85,B 0,C 180,E1 -15584.615,E2 -15584.615} C_VEL
LIN {X 0,Y 314.38,Z 571.597,A -85,B 0,C 180,E1 -15586.16,E2 -15586.16} C_VEL
LIN {X 0,Y 315.442,Z 560.653,A -85,B 0,C 180,E1 -15587.504,E2 -15587.504} C_VEL
LIN {X 0,Y 315.481,Z 555.996,A -85,B 0,C 180,E1 -15588.005,E2 -15588.005} C_VEL
LIN {X 0,Y 314.14,Z 542.475,A -85,B 0,C 180,E1 -15589.268,E2 -15589.268} C_VEL
LIN {X 0,Y 312.593,Z 527.966,A -85,B 0,C 180,E1 -15590.3,E2 -15590.3} C_VEL
LIN {X 0,Y 311.576,Z 517.786,A -85,B 0,C 180,E1 -15590.852,E2 -15590.852} C_VEL
LIN {X 0,Y 312.179,Z 511.29,A -85,B 0,C 180,E1 -15594.613,E2 -15594.613} C_VEL
LIN {X 0,Y 313.119,Z 503.94,A -85,B 0,C 180,E1 -15598.912,E2 -15598.912} C_VEL
LIN {X 0,Y 314.118,Z 496.689,A -85,B 0,C 180,E1 -15603.241,E2 -15603.241} C_VEL
LIN {X 0,Y 314.696,Z 492.97,A -85,B 0,C 180,E1 -15605.496,E2 -15605.496} C_VEL
LIN {X 0,Y 314.643,Z 489.31,A -85,B 0,C 180,E1 -15607.793,E2 -15607.793} C_VEL
LIN {X 0,Y 313.706,Z 483.937,A -85,B 0,C 180,E1 -15611.368,E2 -15611.368} C_VEL
LIN {X 0,Y 312.616,Z 477.546,A -85,B 0,C 180,E1 -15615.82,E2 -15615.82} C_VEL
LIN {X 0,Y 312.531,Z 477.552,A -85,B 0,C 180,E1 -15619.869,E2 -15619.869} C_VEL
LIN {X 0,Y 312.54,Z 477.555,A -85,B 0,C 180,E1 -15622.617,E2 -15622.617} C_VEL
LIN {X 0,Y 312.52,Z 477.555,A -85,B 0,C 180,E1 -15626.311,E2 -15626.311} C_VEL
LIN {X 0,Y 312.539,Z 477.553,A -85,B 0,C 180,E1 -15630.349,E2 -15630.349} C_VEL
LIN {X 0,Y 312.597,Z 477.544,A -85,B 0,C 180,E1 -15634.067,E2 -15634.067} C_VEL
LIN {X 0,Y 312.588,Z 477.544,A -85,B 0,C 180,E1 -15637.529,E2 -15637.529} C_VEL
LIN {X 0,Y 312.639,Z 477.538,A -85,B 0,C 180,E1 -15641.657,E2 -15641.657} C_VEL
LIN {X 0,Y 312.695,Z 477.531,A -85,B 0,C 180,E1 -15645.686,E2 -15645.686} C_VEL
LIN {X 0,Y 312.703,Z 477.53,A -85,B 0,C 180,E1 -15649.642,E2 -15649.642} C_VEL
LIN {X 0,Y 312.873,Z 477.512,A -85,B 0,C 180,E1 -15652.254,E2 -15652.254} C_VEL
LIN {X 0,Y 312.719,Z 477.531,A -85,B 0,C 180,E1 -15654.843,E2 -15654.843} C_VEL
LIN {X 0,Y 312.992,Z 477.498,A -85,B 0,C 180,E1 -15658.714,E2 -15658.714} C_VEL
LIN {X 0,Y 312.993,Z 477.494,A -85,B 0,C 180,E1 -15661.287,E2 -15661.287} C_VEL
LIN {X 0,Y 312.719,Z 477.529,A -85,B 0,C 180,E1 -15665.158,E2 -15665.158} C_VEL
LIN {X 0,Y 312.874,Z 477.509,A -85,B 0,C 180,E1 -15667.746,E2 -15667.746} C_VEL
LIN {X 0,Y 312.671,Z 477.534,A -85,B 0,C 180,E1 -15671.672,E2 -15671.672} C_VEL
LIN {X 0,Y 312.702,Z 477.532,A -85,B 0,C 180,E1 -15674.888,E2 -15674.888} C_VEL
LIN {X 0,Y 312.632,Z 477.539,A -85,B 0,C 180,E1 -15679.237,E2 -15679.237} C_VEL
LIN {X 0,Y 312.548,Z 477.551,A -85,B 0,C 180,E1 -15682.79,E2 -15682.79} C_VEL
LIN {X 0,Y 312.605,Z 477.544,A -85,B 0,C 180,E1 -15685.936,E2 -15685.936} C_VEL
LIN {X 0,Y 312.547,Z 477.55,A -85,B 0,C 180,E1 -15689.65,E2 -15689.65} C_VEL
LIN {X 0,Y 312.521,Z 477.553,A -85,B 0,C 180,E1 -15693.689,E2 -15693.689} C_VEL
LIN {X 0,Y 312.528,Z 477.552,A -85,B 0,C 180,E1 -15697.385,E2 -15697.385} C_VEL
LIN {X 0,Y 312.492,Z 477.558,A -85,B 0,C 180,E1 -15700.709,E2 -15700.709} C_VEL
LIN {X 0,Y 312.454,Z 477.566,A -85,B 0,C 180,E1 -15704.21,E2 -15704.21} C_VEL
LIN {X 0,Y 312.486,Z 477.56,A -85,B 0,C 180,E1 -15707.919,E2 -15707.919} C_VEL
LIN {X 0,Y 312.538,Z 477.553,A -85,B 0,C 180,E1 -15711.911,E2 -15711.911} C_VEL
LIN {X 0,Y 312.509,Z 477.556,A -85,B 0,C 180,E1 -15715.79,E2 -15715.79} C_VEL
LIN {X 0,Y 312.524,Z 477.553,A -85,B 0,C 180,E1 -15718.854,E2 -15718.854} C_VEL
LIN {X 0,Y 312.573,Z 477.549,A -85,B 0,C 180,E1 -15721.825,E2 -15721.825} C_VEL
LIN {X 0,Y 312.589,Z 477.545,A -85,B 0,C 180,E1 -15724.711,E2 -15724.711} C_VEL
LIN {X 0,Y 312.591,Z 477.545,A -85,B 0,C 180,E1 -15727.529,E2 -15727.529} C_VEL
LIN {X 0,Y 312.642,Z 477.54,A -85,B 0,C 180,E1 -15731.657,E2 -15731.657} C_VEL
LIN {X 0,Y 312.698,Z 477.533,A -85,B 0,C 180,E1 -15735.686,E2 -15735.686} C_VEL
LIN {X 0,Y 312.702,Z 477.532,A -85,B 0,C 180,E1 -15739.642,E2 -15739.642} C_VEL
LIN {X 0,Y 312.822,Z 477.519,A -85,B 0,C 180,E1 -15742.253,E2 -15742.253} C_VEL
LIN {X 0,Y 312.711,Z 477.529,A -85,B 0,C 180,E1 -15744.842,E2 -15744.842} C_VEL
LIN {X 0,Y 312.995,Z 477.494,A -85,B 0,C 180,E1 -15748.714,E2 -15748.714} C_VEL
LIN {X 0,Y 312.993,Z 477.495,A -85,B 0,C 180,E1 -15751.287,E2 -15751.287} C_VEL
LIN {X 0,Y 312.719,Z 477.528,A -85,B 0,C 180,E1 -15755.158,E2 -15755.158} C_VEL
LIN {X 0,Y 312.857,Z 477.515,A -85,B 0,C 180,E1 -15757.746,E2 -15757.746} C_VEL
LIN {X 0,Y 312.674,Z 477.537,A -85,B 0,C 180,E1 -15761.671,E2 -15761.671} C_VEL
LIN {X 0,Y 312.704,Z 477.53,A -85,B 0,C 180,E1 -15764.888,E2 -15764.888} C_VEL
LIN {X 0,Y 312.635,Z 477.539,A -85,B 0,C 180,E1 -15769.237,E2 -15769.237} C_VEL
LIN {X 0,Y 312.55,Z 477.549,A -85,B 0,C 180,E1 -15772.789,E2 -15772.789} C_VEL
LIN {X 0,Y 312.606,Z 477.547,A -85,B 0,C 180,E1 -15775.936,E2 -15775.936} C_VEL
LIN {X 0,Y 312.542,Z 477.554,A -85,B 0,C 180,E1 -15779.651,E2 -15779.651} C_VEL
LIN {X 0,Y 312.523,Z 477.557,A -85,B 0,C 180,E1 -15783.689,E2 -15783.689} C_VEL
LIN {X 0,Y 312.541,Z 477.552,A -85,B 0,C 180,E1 -15787.383,E2 -15787.383} C_VEL
LIN {X 0,Y 312.493,Z 477.556,A -85,B 0,C 180,E1 -15790.709,E2 -15790.709} C_VEL
LIN {X 0,Y 312.455,Z 477.563,A -85,B 0,C 180,E1 -15794.209,E2 -15794.209} C_VEL
LIN {X 0,Y 312.487,Z 477.561,A -85,B 0,C 180,E1 -15797.918,E2 -15797.918} C_VEL
LIN {X 0,Y 312.479,Z 477.558,A -85,B 0,C 180,E1 -15800.968,E2 -15800.968} C_VEL
LIN {X 0,Y 312.404,Z 477.569,A -85,B 0,C 180,E1 -15804.203,E2 -15804.203} C_VEL
LIN {X 0,Y 312.09,Z 477.608,A -85,B 0,C 180,E1 -15807.285,E2 -15807.285} C_VEL
LIN {X 0,Y 311.801,Z 477.643,A -85,B 0,C 180,E1 -15810.272,E2 -15810.272} C_VEL
LIN {X 0,Y 311.501,Z 477.685,A -85,B 0,C 180,E1 -15813.177,E2 -15813.177} C_VEL
LIN {X 0,Y 311.385,Z 478.237,A -85,B 0,C 180,E1 -15814.606,E2 -15814.606} C_VEL
LIN {X 0,Y 311.239,Z 482.088,A -85,B 0,C 180,E1 -15818.82,E2 -15818.82} C_VEL
LIN {X 0,Y 311.24,Z 482.745,A -85,B 0,C 180,E1 -15819.404,E2 -15819.404} C_VEL
LIN {X 0,Y 313.734,Z 495.489,A -85,B 0,C 180,E1 -15820.195,E2 -15820.195} C_VEL
LIN {X 0,Y 316.41,Z 509.363,A -85,B 0,C 180,E1 -15821.323,E2 -15821.323} C_VEL
LIN {X 0,Y 316.934,Z 512.223,A -85,B 0,C 180,E1 -15821.595,E2 -15821.595} C_VEL
LIN {X 0,Y 316.065,Z 524.011,A -85,B 0,C 180,E1 -15822.763,E2 -15822.763} C_VEL
LIN {X 0,Y 315.126,Z 535.271,A -85,B 0,C 180,E1 -15824.153,E2 -15824.153} C_VEL
LIN {X 0,Y 314.076,Z 545.802,A -85,B 0,C 180,E1 -15825.75,E2 -15825.75} C_VEL
LIN {X 0,Y 313.462,Z 551.563,A -85,B 0,C 180,E1 -15826.772,E2 -15826.772} C_VEL
LIN {X 0,Y 312.38,Z 555.585,A -85,B 0,C 180,E1 -15827.553,E2 -15827.553} C_VEL
LIN {X 0,Y 308.925,Z 561.632,A -85,B 0,C 180,E1 -15828.852,E2 -15828.852} C_VEL
LIN {X 0,Y 305.575,Z 567.2,A -85,B 0,C 180,E1 -15830.253,E2 -15830.253} C_VEL
LIN {X 0,Y 304.672,Z 570.31,A -85,B 0,C 180,E1 -15831.181,E2 -15831.181} C_VEL
LIN {X 0,Y 304.242,Z 576.51,A -85,B 0,C 180,E1 -15833.367,E2 -15833.367} C_VEL
LIN {X 0,Y 304.067,Z 580.92,A -85,B 0,C 180,E1 -15835.36,E2 -15835.36} C_VEL
LIN {X 0,Y 303.883,Z 584.255,A -85,B 0,C 180,E1 -15837.349,E2 -15837.349} C_VEL
LIN {X 0,Y 303.854,Z 585.942,A -85,B 0,C 180,E1 -15838.674,E2 -15838.674} C_VEL
LIN {X 0,Y 304.02,Z 588.002,A -85,B 0,C 180,E1 -15841.324,E2 -15841.324} C_VEL
LIN {X 0,Y 304.211,Z 588.444,A -85,B 0,C 180,E1 -15842.648,E2 -15842.648} C_VEL
LIN {X 0,Y 304.48,Z 588.472,A -85,B 0,C 180,E1 -15843.97,E2 -15843.97} C_VEL
LIN {X 0,Y 304.678,Z 588.092,A -85,B 0,C 180,E1 -15845.294,E2 -15845.294} C_VEL
LIN {X 0,Y 304.861,Z 587.344,A -85,B 0,C 180,E1 -15846.619,E2 -15846.619} C_VEL
LIN {X 0,Y 305.989,Z 584.906,A -85,B 0,C 180,E1 -15849.02,E2 -15849.02} C_VEL
LIN {X 0,Y 307.15,Z 581.486,A -85,B 0,C 180,E1 -15851.215,E2 -15851.215} C_VEL
LIN {X 0,Y 308.597,Z 577.344,A -85,B 0,C 180,E1 -15853.164,E2 -15853.164} C_VEL
LIN {X 0,Y 310.583,Z 571.088,A -85,B 0,C 180,E1 -15855.419,E2 -15855.419} C_VEL
LIN {X 0,Y 312.983,Z 563.274,A -85,B 0,C 180,E1 -15857.646,E2 -15857.646} C_VEL
LIN {X 0,Y 315.629,Z 554.808,A -85,B 0,C 180,E1 -15859.512,E2 -15859.512} C_VEL
LIN {X 0,Y 318.443,Z 544.631,A -85,B 0,C 180,E1 -15861.355,E2 -15861.355} C_VEL
LIN {X 0,Y 321.08,Z 534.244,A -85,B 0,C 180,E1 -15862.867,E2 -15862.867} C_VEL
LIN {X 0,Y 321.914,Z 530.817,A -85,B 0,C 180,E1 -15863.3,E2 -15863.3} C_VEL
LIN {X 0,Y 321.972,Z 529.233,A -85,B 0,C 180,E1 -15863.54,E2 -15863.54} C_VEL
LIN {X 0,Y 320.039,Z 520.957,A -85,B 0,C 180,E1 -15865.147,E2 -15865.147} C_VEL
LIN {X 0,Y 317.162,Z 512.632,A -85,B 0,C 180,E1 -15866.886,E2 -15866.886} C_VEL
LIN {X 0,Y 313.717,Z 505.464,A -85,B 0,C 180,E1 -15868.619,E2 -15868.619} C_VEL
LIN {X 0,Y 312.139,Z 502.391,A -85,B 0,C 180,E1 -15869.403,E2 -15869.403} C_VEL
LIN {X 0,Y 310.81,Z 500.473,A -85,B 0,C 180,E1 -15870.002,E2 -15870.002} C_VEL
LIN {X 0,Y 309.969,Z 498.419,A -85,B 0,C 180,E1 -15870.505,E2 -15870.505} C_VEL
LIN {X 0,Y 308.438,Z 496.798,A -85,B 0,C 180,E1 -15871.171,E2 -15871.171} C_VEL
LIN {X 0,Y 307.198,Z 493.803,A -85,B 0,C 180,E1 -15871.944,E2 -15871.944} C_VEL
LIN {X 0,Y 307.626,Z 493.647,A -85,B 0,C 180,E1 -15874.83,E2 -15874.83} C_VEL
LIN {X 0,Y 308.04,Z 493.896,A -85,B 0,C 180,E1 -15878.025,E2 -15878.025} C_VEL
LIN {X 0,Y 308.325,Z 494.7,A -85,B 0,C 180,E1 -15881.378,E2 -15881.378} C_VEL
LIN {X 0,Y 308.648,Z 496.255,A -85,B 0,C 180,E1 -15885.099,E2 -15885.099} C_VEL
LIN {X 0,Y 308.983,Z 498.48,A -85,B 0,C 180,E1 -15888.729,E2 -15888.729} C_VEL
LIN {X 0,Y 309.151,Z 499.928,A -85,B 0,C 180,E1 -15890.618,E2 -15890.618} C_VEL
LIN {X 0,Y 309.056,Z 501.839,A -85,B 0,C 180,E1 -15892.741,E2 -15892.741} C_VEL
LIN {X 0,Y 308.487,Z 504.522,A -85,B 0,C 180,E1 -15895.281,E2 -15895.281} C_VEL
LIN {X 0,Y 307.643,Z 507.914,A -85,B 0,C 180,E1 -15898.098,E2 -15898.098} C_VEL
LIN {X 0,Y 308.407,Z 511.227,A -85,B 0,C 180,E1 -15898.676,E2 -15898.676} C_VEL
LIN {X 0,Y 309.568,Z 513.591,A -85,B 0,C 180,E1 -15899.246,E2 -15899.246} C_VEL
LIN {X 0,Y 313.506,Z 526.566,A -85,B 0,C 180,E1 -15901.581,E2 -15901.581} C_VEL
LIN {X 0,Y 315.851,Z 537.082,A -85,B 0,C 180,E1 -15903.287,E2 -15903.287} C_VEL
LIN {X 0,Y 317.189,Z 547.772,A -85,B 0,C 180,E1 -15904.903,E2 -15904.903} C_VEL
LIN {X 0,Y 317.342,Z 558.689,A -85,B 0,C 180,E1 -15906.507,E2 -15906.507} C_VEL
LIN {X 0,Y 316.073,Z 568.507,A -85,B 0,C 180,E1 -15907.962,E2 -15907.962} C_VEL
LIN {X 0,Y 313.387,Z 579.224,A -85,B 0,C 180,E1 -15909.659,E2 -15909.659} C_VEL
LIN {X 0,Y 310.8,Z 588.882,A -85,B 0,C 180,E1 -15911.544,E2 -15911.544} C_VEL
LIN {X 0,Y 308.531,Z 597.229,A -85,B 0,C 180,E1 -15913.531,E2 -15913.531} C_VEL
LIN {X 0,Y 307.03,Z 603.684,A -85,B 0,C 180,E1 -15915.416,E2 -15915.416} C_VEL
LIN {X 0,Y 305.575,Z 609.215,A -85,B 0,C 180,E1 -15917.379,E2 -15917.379} C_VEL
LIN {X 0,Y 304.678,Z 613.681,A -85,B 0,C 180,E1 -15919.366,E2 -15919.366} C_VEL
LIN {X 0,Y 304.274,Z 616.126,A -85,B 0,C 180,E1 -15920.695,E2 -15920.695} C_VEL
LIN {X 0,Y 303.953,Z 618.106,A -85,B 0,C 180,E1 -15922.025,E2 -15922.025} C_VEL
LIN {X 0,Y 303.686,Z 620.843,A -85,B 0,C 180,E1 -15924.688,E2 -15924.688} C_VEL
LIN {X 0,Y 303.736,Z 621.631,A -85,B 0,C 180,E1 -15926.019,E2 -15926.019} C_VEL
LIN {X 0,Y 303.736,Z 621.979,A -85,B 0,C 180,E1 -15927.347,E2 -15927.347} C_VEL
LIN {X 0,Y 303.937,Z 621.91,A -85,B 0,C 180,E1 -15928.675,E2 -15928.675} C_VEL
LIN {X 0,Y 304.049,Z 621.426,A -85,B 0,C 180,E1 -15930,E2 -15930} C_VEL
LIN {X 0,Y 304.055,Z 620.52,A -85,B 0,C 180,E1 -15931.324,E2 -15931.324} C_VEL
LIN {X 0,Y 303.884,Z 619.13,A -85,B 0,C 180,E1 -15932.651,E2 -15932.651} C_VEL
LIN {X 0,Y 303.94,Z 616.221,A -85,B 0,C 180,E1 -15934.642,E2 -15934.642} C_VEL
LIN {X 0,Y 304.02,Z 612.187,A -85,B 0,C 180,E1 -15936.637,E2 -15936.637} C_VEL
LIN {X 0,Y 304.239,Z 605.923,A -85,B 0,C 180,E1 -15938.97,E2 -15938.97} C_VEL
LIN {X 0,Y 304.654,Z 599.081,A -85,B 0,C 180,E1 -15940.971,E2 -15940.971} C_VEL
LIN {X 0,Y 305.443,Z 590.561,A -85,B 0,C 180,E1 -15942.964,E2 -15942.964} C_VEL
LIN {X 0,Y 306.385,Z 580.127,A -85,B 0,C 180,E1 -15944.931,E2 -15944.931} C_VEL
LIN {X 0,Y 307.546,Z 569.492,A -85,B 0,C 180,E1 -15946.529,E2 -15946.529} C_VEL
LIN {X 0,Y 308.542,Z 558.2,A -85,B 0,C 180,E1 -15947.909,E2 -15947.909} C_VEL
LIN {X 0,Y 307.451,Z 546.472,A -85,B 0,C 180,E1 -15949.101,E2 -15949.101} C_VEL
LIN {X 0,Y 306.008,Z 532.318,A -85,B 0,C 180,E1 -15950.239,E2 -15950.239} C_VEL
LIN {X 0,Y 304.548,Z 518.232,A -85,B 0,C 180,E1 -15951.069,E2 -15951.069} C_VEL
LIN {X 0,Y 304.536,Z 517.404,A -85,B 0,C 180,E1 -15951.136,E2 -15951.136} C_VEL
LIN {X 0,Y 305.189,Z 510.567,A -85,B 0,C 180,E1 -15955.215,E2 -15955.215} C_VEL
LIN {X 0,Y 306.111,Z 503.854,A -85,B 0,C 180,E1 -15959.256,E2 -15959.256} C_VEL
LIN {X 0,Y 307.243,Z 496.189,A -85,B 0,C 180,E1 -15963.959,E2 -15963.959} C_VEL
LIN {X 0,Y 307.688,Z 492.258,A -85,B 0,C 180,E1 -15966.432,E2 -15966.432} C_VEL
LIN {X 0,Y 307.29,Z 488.433,A -85,B 0,C 180,E1 -15968.958,E2 -15968.958} C_VEL
LIN {X 0,Y 306.319,Z 482.896,A -85,B 0,C 180,E1 -15972.761,E2 -15972.761} C_VEL
LIN {X 0,Y 305.565,Z 478.423,A -85,B 0,C 180,E1 -15976.137,E2 -15976.137} C_VEL
LIN {X 0,Y 305.484,Z 478.43,A -85,B 0,C 180,E1 -15979.897,E2 -15979.897} C_VEL
LIN {X 0,Y 305.5,Z 478.427,A -85,B 0,C 180,E1 -15983.627,E2 -15983.627} C_VEL
LIN {X 0,Y 305.466,Z 478.435,A -85,B 0,C 180,E1 -15986.483,E2 -15986.483} C_VEL
LIN {X 0,Y 305.458,Z 478.433,A -85,B 0,C 180,E1 -15989.591,E2 -15989.591} C_VEL
LIN {X 0,Y 305.515,Z 478.43,A -85,B 0,C 180,E1 -15992.608,E2 -15992.608} C_VEL
LIN {X 0,Y 305.509,Z 478.427,A -85,B 0,C 180,E1 -15995.539,E2 -15995.539} C_VEL
LIN {X 0,Y 305.521,Z 478.425,A -85,B 0,C 180,E1 -15999.815,E2 -15999.815} C_VEL
LIN {X 0,Y 305.576,Z 478.423,A -85,B 0,C 180,E1 -16002.603,E2 -16002.603} C_VEL
LIN {X 0,Y 305.65,Z 478.409,A -85,B 0,C 180,E1 -16005.349,E2 -16005.349} C_VEL
LIN {X 0,Y 305.64,Z 478.41,A -85,B 0,C 180,E1 -16009.4,E2 -16009.4} C_VEL
LIN {X 0,Y 305.814,Z 478.39,A -85,B 0,C 180,E1 -16012.075,E2 -16012.075} C_VEL
LIN {X 0,Y 305.69,Z 478.407,A -85,B 0,C 180,E1 -16014.724,E2 -16014.724} C_VEL
LIN {X 0,Y 305.959,Z 478.374,A -85,B 0,C 180,E1 -16018.684,E2 -16018.684} C_VEL
LIN {X 0,Y 305.959,Z 478.37,A -85,B 0,C 180,E1 -16021.316,E2 -16021.316} C_VEL
LIN {X 0,Y 305.852,Z 478.387,A -85,B 0,C 180,E1 -16026.617,E2 -16026.617} C_VEL
LIN {X 0,Y 305.737,Z 478.398,A -85,B 0,C 180,E1 -16029.26,E2 -16029.26} C_VEL
LIN {X 0,Y 305.591,Z 478.416,A -85,B 0,C 180,E1 -16033.296,E2 -16033.296} C_VEL
LIN {X 0,Y 305.595,Z 478.417,A -85,B 0,C 180,E1 -16036.02,E2 -16036.02} C_VEL
LIN {X 0,Y 305.579,Z 478.418,A -85,B 0,C 180,E1 -16039.446,E2 -16039.446} C_VEL
LIN {X 0,Y 305.492,Z 478.429,A -85,B 0,C 180,E1 -16043.042,E2 -16043.042} C_VEL
LIN {X 0,Y 305.549,Z 478.425,A -85,B 0,C 180,E1 -16046.227,E2 -16046.227} C_VEL
LIN {X 0,Y 305.497,Z 478.428,A -85,B 0,C 180,E1 -16049.05,E2 -16049.05} C_VEL
LIN {X 0,Y 305.446,Z 478.436,A -85,B 0,C 180,E1 -16051.952,E2 -16051.952} C_VEL
LIN {X 0,Y 305.464,Z 478.432,A -85,B 0,C 180,E1 -16055.113,E2 -16055.113} C_VEL
LIN {X 0,Y 305.469,Z 478.435,A -85,B 0,C 180,E1 -16058.533,E2 -16058.533} C_VEL
LIN {X 0,Y 305.457,Z 478.435,A -85,B 0,C 180,E1 -16062.586,E2 -16062.586} C_VEL
LIN {X 0,Y 305.428,Z 478.441,A -85,B 0,C 180,E1 -16066.345,E2 -16066.345} C_VEL
LIN {X 0,Y 305.46,Z 478.435,A -85,B 0,C 180,E1 -16069.893,E2 -16069.893} C_VEL
LIN {X 0,Y 305.502,Z 478.428,A -85,B 0,C 180,E1 -16073.627,E2 -16073.627} C_VEL
LIN {X 0,Y 305.468,Z 478.434,A -85,B 0,C 180,E1 -16076.484,E2 -16076.484} C_VEL
LIN {X 0,Y 305.461,Z 478.433,A -85,B 0,C 180,E1 -16079.591,E2 -16079.591} C_VEL
LIN {X 0,Y 305.522,Z 478.427,A -85,B 0,C 180,E1 -16082.609,E2 -16082.609} C_VEL
LIN {X 0,Y 305.511,Z 478.427,A -85,B 0,C 180,E1 -16085.539,E2 -16085.539} C_VEL
LIN {X 0,Y 305.523,Z 478.427,A -85,B 0,C 180,E1 -16089.815,E2 -16089.815} C_VEL
LIN {X 0,Y 305.578,Z 478.419,A -85,B 0,C 180,E1 -16092.603,E2 -16092.603} C_VEL
LIN {X 0,Y 305.653,Z 478.409,A -85,B 0,C 180,E1 -16095.349,E2 -16095.349} C_VEL
LIN {X 0,Y 305.639,Z 478.411,A -85,B 0,C 180,E1 -16099.4,E2 -16099.4} C_VEL
LIN {X 0,Y 305.769,Z 478.399,A -85,B 0,C 180,E1 -16102.073,E2 -16102.073} C_VEL
LIN {X 0,Y 305.68,Z 478.405,A -85,B 0,C 180,E1 -16104.723,E2 -16104.723} C_VEL
LIN {X 0,Y 305.962,Z 478.371,A -85,B 0,C 180,E1 -16108.684,E2 -16108.684} C_VEL
LIN {X 0,Y 305.96,Z 478.371,A -85,B 0,C 180,E1 -16111.316,E2 -16111.316} C_VEL
LIN {X 0,Y 305.69,Z 478.404,A -85,B 0,C 180,E1 -16115.277,E2 -16115.277} C_VEL
LIN {X 0,Y 305.801,Z 478.395,A -85,B 0,C 180,E1 -16117.926,E2 -16117.926} C_VEL
LIN {X 0,Y 305.608,Z 478.419,A -85,B 0,C 180,E1 -16121.945,E2 -16121.945} C_VEL
LIN {X 0,Y 305.642,Z 478.41,A -85,B 0,C 180,E1 -16125.035,E2 -16125.035} C_VEL
LIN {X 0,Y 305.581,Z 478.419,A -85,B 0,C 180,E1 -16129.445,E2 -16129.445} C_VEL
LIN {X 0,Y 305.494,Z 478.428,A -85,B 0,C 180,E1 -16133.041,E2 -16133.041} C_VEL
LIN {X 0,Y 305.535,Z 478.425,A -85,B 0,C 180,E1 -16136.221,E2 -16136.221} C_VEL
LIN {X 0,Y 305.491,Z 478.429,A -85,B 0,C 180,E1 -16139.047,E2 -16139.047} C_VEL
LIN {X 0,Y 305.447,Z 478.438,A -85,B 0,C 180,E1 -16141.952,E2 -16141.952} C_VEL
LIN {X 0,Y 305.466,Z 478.432,A -85,B 0,C 180,E1 -16145.113,E2 -16145.113} C_VEL
LIN {X 0,Y 305.47,Z 478.431,A -85,B 0,C 180,E1 -16148.533,E2 -16148.533} C_VEL
LIN {X 0,Y 305.458,Z 478.433,A -85,B 0,C 180,E1 -16152.586,E2 -16152.586} C_VEL
LIN {X 0,Y 305.429,Z 478.437,A -85,B 0,C 180,E1 -16156.345,E2 -16156.345} C_VEL
LIN {X 0,Y 305.46,Z 478.436,A -85,B 0,C 180,E1 -16159.892,E2 -16159.892} C_VEL
LIN {X 0,Y 305.385,Z 478.447,A -85,B 0,C 180,E1 -16163.657,E2 -16163.657} C_VEL
LIN {X 0,Y 305.136,Z 478.473,A -85,B 0,C 180,E1 -16166.442,E2 -16166.442} C_VEL
LIN {X 0,Y 304.828,Z 478.515,A -85,B 0,C 180,E1 -16169.52,E2 -16169.52} C_VEL
LIN {X 0,Y 304.522,Z 478.557,A -85,B 0,C 180,E1 -16172.511,E2 -16172.511} C_VEL
LIN {X 0,Y 304.328,Z 478.589,A -85,B 0,C 180,E1 -16174.244,E2 -16174.244} C_VEL
LIN {X 0,Y 304.173,Z 482.234,A -85,B 0,C 180,E1 -16178.303,E2 -16178.303} C_VEL
LIN {X 0,Y 304.18,Z 483.216,A -85,B 0,C 180,E1 -16179.148,E2 -16179.148} C_VEL
LIN {X 0,Y 306.686,Z 496.131,A -85,B 0,C 180,E1 -16179.978,E2 -16179.978} C_VEL
LIN {X 0,Y 309.152,Z 508.838,A -85,B 0,C 180,E1 -16181.036,E2 -16181.036} C_VEL
LIN {X 0,Y 309.918,Z 513.566,A -85,B 0,C 180,E1 -16181.489,E2 -16181.489} C_VEL
LIN {X 0,Y 309.017,Z 524.72,A -85,B 0,C 180,E1 -16182.632,E2 -16182.632} C_VEL
LIN {X 0,Y 308.016,Z 536.298,A -85,B 0,C 180,E1 -16184.109,E2 -16184.109} C_VEL
LIN {X 0,Y 306.933,Z 546.781,A -85,B 0,C 180,E1 -16185.75,E2 -16185.75} C_VEL
LIN {X 0,Y 306.038,Z 555.468,A -85,B 0,C 180,E1 -16187.399,E2 -16187.399} C_VEL
LIN {X 0,Y 305.243,Z 563.998,A -85,B 0,C 180,E1 -16189.386,E2 -16189.386} C_VEL
LIN {X 0,Y 304.672,Z 570.31,A -85,B 0,C 180,E1 -16191.181,E2 -16191.181} C_VEL
LIN {X 0,Y 303.818,Z 573.236,A -85,B 0,C 180,E1 -16192.137,E2 -16192.137} C_VEL
LIN {X 0,Y 300.713,Z 577.493,A -85,B 0,C 180,E1 -16193.729,E2 -16193.729} C_VEL
LIN {X 0,Y 297.643,Z 581.147,A -85,B 0,C 180,E1 -16195.405,E2 -16195.405} C_VEL
LIN {X 0,Y 296.865,Z 583.076,A -85,B 0,C 180,E1 -16196.475,E2 -16196.475} C_VEL
LIN {X 0,Y 296.762,Z 586.097,A -85,B 0,C 180,E1 -16198.643,E2 -16198.643} C_VEL
LIN {X 0,Y 296.804,Z 587.445,A -85,B 0,C 180,E1 -16200,E2 -16200} C_VEL
LIN {X 0,Y 297.131,Z 588.869,A -85,B 0,C 180,E1 -16202.711,E2 -16202.711} C_VEL
LIN {X 0,Y 297.409,Z 589.003,A -85,B 0,C 180,E1 -16204.065,E2 -16204.065} C_VEL
LIN {X 0,Y 297.624,Z 588.742,A -85,B 0,C 180,E1 -16205.42,E2 -16205.42} C_VEL
LIN {X 0,Y 297.848,Z 588.069,A -85,B 0,C 180,E1 -16206.775,E2 -16206.775} C_VEL
LIN {X 0,Y 299.174,Z 585.548,A -85,B 0,C 180,E1 -16209.464,E2 -16209.464} C_VEL
LIN {X 0,Y 300.277,Z 582.587,A -85,B 0,C 180,E1 -16211.475,E2 -16211.475} C_VEL
LIN {X 0,Y 301.801,Z 578.618,A -85,B 0,C 180,E1 -16213.466,E2 -16213.466} C_VEL
LIN {X 0,Y 303.593,Z 573.65,A -85,B 0,C 180,E1 -16215.439,E2 -16215.439} C_VEL
LIN {X 0,Y 306.042,Z 566.338,A -85,B 0,C 180,E1 -16217.714,E2 -16217.714} C_VEL
LIN {X 0,Y 309.232,Z 557.111,A -85,B 0,C 180,E1 -16219.932,E2 -16219.932} C_VEL
LIN {X 0,Y 312.194,Z 547.342,A -85,B 0,C 180,E1 -16221.804,E2 -16221.804} C_VEL
LIN {X 0,Y 314.941,Z 537.5,A -85,B 0,C 180,E1 -16223.339,E2 -16223.339} C_VEL
LIN {X 0,Y 316.091,Z 533.172,A -85,B 0,C 180,E1 -16223.927,E2 -16223.927} C_VEL
LIN {X 0,Y 316.09,Z 531.203,A -85,B 0,C 180,E1 -16224.272,E2 -16224.272} C_VEL
LIN {X 0,Y 313.723,Z 521.408,A -85,B 0,C 180,E1 -16226.352,E2 -16226.352} C_VEL
LIN {X 0,Y 311.597,Z 515.594,A -85,B 0,C 180,E1 -16227.714,E2 -16227.714} C_VEL
LIN {X 0,Y 307.903,Z 507.657,A -85,B 0,C 180,E1 -16229.845,E2 -16229.845} C_VEL
LIN {X 0,Y 305.986,Z 503.914,A -85,B 0,C 180,E1 -16230.968,E2 -16230.968} C_VEL
LIN {X 0,Y 304.316,Z 501.577,A -85,B 0,C 180,E1 -16231.856,E2 -16231.856} C_VEL
LIN {X 0,Y 303.929,Z 500.633,A -85,B 0,C 180,E1 -16232.13,E2 -16232.13} C_VEL
LIN {X 0,Y 301.23,Z 497.121,A -85,B 0,C 180,E1 -16233.683,E2 -16233.683} C_VEL
LIN {X 0,Y 300.592,Z 495.216,A -85,B 0,C 180,E1 -16234.26,E2 -16234.26} C_VEL
LIN {X 0,Y 301.052,Z 495.412,A -85,B 0,C 180,E1 -16237.465,E2 -16237.465} C_VEL
LIN {X 0,Y 301.357,Z 496.127,A -85,B 0,C 180,E1 -16240.768,E2 -16240.768} C_VEL
LIN {X 0,Y 301.613,Z 497.503,A -85,B 0,C 180,E1 -16244.35,E2 -16244.35} C_VEL
LIN {X 0,Y 301.978,Z 499.651,A -85,B 0,C 180,E1 -16248.137,E2 -16248.137} C_VEL
LIN {X 0,Y 302.184,Z 501.88,A -85,B 0,C 180,E1 -16251.101,E2 -16251.101} C_VEL
